   1:  PR[GP1:91,2] = PR[GP1:90,2] + -1.651;
   1:L PR[91] R[100]mm/sec CNT100;
   1:  PR[GP1:91,1] = PR[GP1:90,1] + -34.835;
   1:  PR[GP1:91,2] = PR[GP1:90,2] + -4.892;
   1:L PR[91] R[100]mm/sec CNT100;
   1:  PR[GP1:91,1] = PR[GP1:90,1] + -34.523;
   1:  PR[GP1:91,2] = PR[GP1:90,2] + -6.094;
   1:L PR[91] R[100]mm/sec CNT100;
   1:  PR[GP1:91,1] = PR[GP1:90,1] + -33.966;
   1:  PR[GP1:91,2] = PR[GP1:90,2] + -7.337;
   1:L PR[91] R[100]mm/sec CNT100;
   1:  PR[GP1:91,1] = PR[GP1:90,1] + -32.585;
   1:  PR[GP1:91,2] = PR[GP1:90,2] + -10.486;
   1:L PR[91] R[100]mm/sec CNT100;
   1:  PR[GP1:91,1] = PR[GP1:90,1] + -31.931;
   1:  PR[GP1:91,2] = PR[GP1:90,2] + -11.478;
   1:L PR[91] R[100]mm/sec CNT100;
   1:  PR[GP1:91,1] = PR[GP1:90,1] + -29.572;
   1:  PR[GP1:91,2] = PR[GP1:90,2] + -14.403;
   1:L PR[91] R[100]mm/sec CNT100;
   1:  PR[GP1:91,1] = PR[GP1:90,1] + -28.833;
   1:  PR[GP1:91,2] = PR[GP1:90,2] + -15.201;
   1:L PR[91] R[100]mm/sec CNT100;
   1:  PR[GP1:91,1] = PR[GP1:90,1] + -28.025;
   1:  PR[GP1:91,2] = PR[GP1:90,2] + -15.834;
   1:L PR[91] R[100]mm/sec CNT100;
   1:  PR[GP1:91,1] = PR[GP1:90,1] + -24.662;
   1:  PR[GP1:91,2] = PR[GP1:90,2] + -18.272;
   1:L PR[91] R[100]mm/sec CNT100;
   1:  PR[GP1:91,1] = PR[GP1:90,1] + -23.931;
   1:  PR[GP1:91,2] = PR[GP1:90,2] + -18.681;
   1:L PR[91] R[100]mm/sec CNT100;
   1:  PR[GP1:91,1] = PR[GP1:90,1] + -23.152;
   1:  PR[GP1:91,2] = PR[GP1:90,2] + -18.969;
   1:L PR[91] R[100]mm/sec CNT100;
   1:  PR[GP1:91,1] = PR[GP1:90,1] + -18.880;
   1:  PR[GP1:91,2] = PR[GP1:90,2] + -20.635;
   1:L PR[91] R[100]mm/sec CNT100;
   1:  PR[GP1:91,1] = PR[GP1:90,1] + -18.320;
   1:  PR[GP1:91,2] = PR[GP1:90,2] + -20.751;
   1:L PR[91] R[100]mm/sec CNT100;
   1:  PR[GP1:91,1] = PR[GP1:90,1] + -13.243;
   1:  PR[GP1:91,2] = PR[GP1:90,2] + -21.342;
   1:L PR[91] R[100]mm/sec CNT100;
   1:  PR[GP1:91,1] = PR[GP1:90,1] + -12.848;
   1:  PR[GP1:91,2] = PR[GP1:90,2] + -21.363;
   1:L PR[91] R[100]mm/sec CNT100;
   1:  PR[GP1:91,1] = PR[GP1:90,1] + -12.498;
   1:  PR[GP1:91,2] = PR[GP1:90,2] + -21.328;
   1:L PR[91] R[100]mm/sec CNT100;
   1:  PR[GP1:91,1] = PR[GP1:90,1] + -7.066;
   1:  PR[GP1:91,2] = PR[GP1:90,2] + -20.567;
   1:L PR[91] R[100]mm/sec CNT100;
   1:  PR[GP1:91,1] = PR[GP1:90,1] + -6.974;
   1:  PR[GP1:91,2] = PR[GP1:90,2] + -20.544;
   1:L PR[91] R[100]mm/sec CNT100;
   1:  PR[GP1:91,1] = PR[GP1:90,1] + -1.723;
   1:  PR[GP1:91,2] = PR[GP1:90,2] + -18.303;
   1:L PR[91] R[100]mm/sec CNT100;
   1:  PR[GP1:91,1] = PR[GP1:90,1] + -1.227;
   1:  PR[GP1:91,2] = PR[GP1:90,2] + -18.103;
   1:L PR[91] R[100]mm/sec CNT100;
   1:  PR[GP1:91,1] = PR[GP1:90,1] + -0.702;
   1:  PR[GP1:91,2] = PR[GP1:90,2] + -17.952;
   1:L PR[91] R[100]mm/sec CNT100;
   1:  PR[GP1:91,1] = PR[GP1:90,1] + 0.096;
   1:  PR[GP1:91,2] = PR[GP1:90,2] + -17.623;
   1:L PR[91] R[100]mm/sec CNT100;
   1:  PR[GP1:91,1] = PR[GP1:90,1] + 1.055;
   1:  PR[GP1:91,2] = PR[GP1:90,2] + -17.917;
   1:L PR[91] R[100]mm/sec CNT100;
   1:  PR[GP1:91,1] = PR[GP1:90,1] + 1.526;
   1:  PR[GP1:91,2] = PR[GP1:90,2] + -18.164;
   1:L PR[91] R[100]mm/sec CNT100;
   1:  PR[GP1:91,1] = PR[GP1:90,1] + 7.126;
   1:  PR[GP1:91,2] = PR[GP1:90,2] + -20.540;
   1:L PR[91] R[100]mm/sec CNT100;
   1:  PR[GP1:91,1] = PR[GP1:90,1] + 7.196;
   1:  PR[GP1:91,2] = PR[GP1:90,2] + -20.559;
   1:L PR[91] R[100]mm/sec CNT100;
   1:  PR[GP1:91,1] = PR[GP1:90,1] + 7.432;
   1:  PR[GP1:91,2] = PR[GP1:90,2] + -20.583;
   1:L PR[91] R[100]mm/sec CNT100;
   1:  PR[GP1:91,1] = PR[GP1:90,1] + 13.029;
   1:  PR[GP1:91,2] = PR[GP1:90,2] + -21.362;
   1:L PR[91] R[100]mm/sec CNT100;
   1:  PR[GP1:91,1] = PR[GP1:90,1] + 13.393;
   1:  PR[GP1:91,2] = PR[GP1:90,2] + -21.343;
   1:L PR[91] R[100]mm/sec CNT100;
   1:  PR[GP1:91,1] = PR[GP1:90,1] + 18.470;
   1:  PR[GP1:91,2] = PR[GP1:90,2] + -20.751;
   1:L PR[91] R[100]mm/sec CNT100;
   1:  PR[GP1:91,1] = PR[GP1:90,1] + 19.041;
   1:  PR[GP1:91,2] = PR[GP1:90,2] + -20.633;
   1:L PR[91] R[100]mm/sec CNT100;
   1:  PR[GP1:91,1] = PR[GP1:90,1] + 19.722;
   1:  PR[GP1:91,2] = PR[GP1:90,2] + -20.382;
   1:L PR[91] R[100]mm/sec CNT100;
   1:  PR[GP1:91,1] = PR[GP1:90,1] + 24.072;
   1:  PR[GP1:91,2] = PR[GP1:90,2] + -18.690;
   1:L PR[91] R[100]mm/sec CNT100;
   1:  PR[GP1:91,1] = PR[GP1:90,1] + 24.789;
   1:  PR[GP1:91,2] = PR[GP1:90,2] + -18.291;
   1:L PR[91] R[100]mm/sec CNT100;
   1:  PR[GP1:91,1] = PR[GP1:90,1] + 25.600;
   1:  PR[GP1:91,2] = PR[GP1:90,2] + -17.662;
   1:L PR[91] R[100]mm/sec CNT100;
   1:  PR[GP1:91,1] = PR[GP1:90,1] + 28.990;
   1:  PR[GP1:91,2] = PR[GP1:90,2] + -15.200;
   1:L PR[91] R[100]mm/sec CNT100;
   1:  PR[GP1:91,1] = PR[GP1:90,1] + 29.712;
   1:  PR[GP1:91,2] = PR[GP1:90,2] + -14.420;
   1:L PR[91] R[100]mm/sec CNT100;
   1:  PR[GP1:91,1] = PR[GP1:90,1] + 32.073;
   1:  PR[GP1:91,2] = PR[GP1:90,2] + -11.489;
   1:L PR[91] R[100]mm/sec CNT100;
   1:  PR[GP1:91,1] = PR[GP1:90,1] + 32.740;
   1:  PR[GP1:91,2] = PR[GP1:90,2] + -10.480;
   1:L PR[91] R[100]mm/sec CNT100;
   1:  PR[GP1:91,1] = PR[GP1:90,1] + 33.295;
   1:  PR[GP1:91,2] = PR[GP1:90,2] + -9.259;
   1:L PR[91] R[100]mm/sec CNT100;
   1:  PR[GP1:91,1] = PR[GP1:90,1] + 34.672;
   1:  PR[GP1:91,2] = PR[GP1:90,2] + -6.135;
   1:L PR[91] R[100]mm/sec CNT100;
   1:  PR[GP1:91,1] = PR[GP1:90,1] + 34.975;
   1:  PR[GP1:91,2] = PR[GP1:90,2] + -4.983;
   1:L PR[91] R[100]mm/sec CNT100;
   1:  PR[GP1:91,1] = PR[GP1:90,1] + 35.092;
   1:  PR[GP1:91,2] = PR[GP1:90,2] + -3.555;
   1:L PR[91] R[100]mm/sec CNT100;
   1:  PR[GP1:91,1] = PR[GP1:90,1] + 35.547;
   1:  PR[GP1:91,2] = PR[GP1:90,2] + -0.271;
   1:L PR[91] R[100]mm/sec CNT100;
   1:  PR[GP1:91,1] = PR[GP1:90,1] + 35.437;
   1:  PR[GP1:91,2] = PR[GP1:90,2] + 1.070;
   1:L PR[91] R[100]mm/sec CNT100;
   1:  PR[GP1:91,1] = PR[GP1:90,1] + 34.986;
   1:  PR[GP1:91,2] = PR[GP1:90,2] + 4.315;
   1:L PR[91] R[100]mm/sec CNT100;
   1:  PR[GP1:91,1] = PR[GP1:90,1] + 34.676;
   1:  PR[GP1:91,2] = PR[GP1:90,2] + 5.499;
   1:L PR[91] R[100]mm/sec CNT100;
   1:  PR[GP1:91,1] = PR[GP1:90,1] + 34.119;
   1:  PR[GP1:91,2] = PR[GP1:90,2] + 6.723;
   1:L PR[91] R[100]mm/sec CNT100;
   1:  PR[GP1:91,1] = PR[GP1:90,1] + 32.741;
   1:  PR[GP1:91,2] = PR[GP1:90,2] + 9.856;
   1:L PR[91] R[100]mm/sec CNT100;
   1:  PR[GP1:91,1] = PR[GP1:90,1] + 32.078;
   1:  PR[GP1:91,2] = PR[GP1:90,2] + 10.857;
   1:L PR[91] R[100]mm/sec CNT100;
   1:  PR[GP1:91,1] = PR[GP1:90,1] + 29.723;
   1:  PR[GP1:91,2] = PR[GP1:90,2] + 13.786;
   1:L PR[91] R[100]mm/sec CNT100;
   1:  PR[GP1:91,1] = PR[GP1:90,1] + 28.984;
   1:  PR[GP1:91,2] = PR[GP1:90,2] + 14.583;
   1:L PR[91] R[100]mm/sec CNT100;
   1:  PR[GP1:91,1] = PR[GP1:90,1] + 28.182;
   1:  PR[GP1:91,2] = PR[GP1:90,2] + 15.208;
   1:L PR[91] R[100]mm/sec CNT100;
   1:  PR[GP1:91,1] = PR[GP1:90,1] + 24.828;
   1:  PR[GP1:91,2] = PR[GP1:90,2] + 17.645;
   1:L PR[91] R[100]mm/sec CNT100;
   1:  PR[GP1:91,1] = PR[GP1:90,1] + 24.103;
   1:  PR[GP1:91,2] = PR[GP1:90,2] + 18.049;
   1:L PR[91] R[100]mm/sec CNT100;
   1:  PR[GP1:91,1] = PR[GP1:90,1] + 23.320;
   1:  PR[GP1:91,2] = PR[GP1:90,2] + 18.337;
   1:L PR[91] R[100]mm/sec CNT100;
   1:  PR[GP1:91,1] = PR[GP1:90,1] + 19.058;
   1:  PR[GP1:91,2] = PR[GP1:90,2] + 20.004;
   1:L PR[91] R[100]mm/sec CNT100;
   1:  PR[GP1:91,1] = PR[GP1:90,1] + 18.498;
   1:  PR[GP1:91,2] = PR[GP1:90,2] + 20.120;
   1:L PR[91] R[100]mm/sec CNT100;
   1:  PR[GP1:91,1] = PR[GP1:90,1] + 13.433;
   1:  PR[GP1:91,2] = PR[GP1:90,2] + 20.719;
   1:L PR[91] R[100]mm/sec CNT100;
   1:  PR[GP1:91,1] = PR[GP1:90,1] + 13.042;
   1:  PR[GP1:91,2] = PR[GP1:90,2] + 20.740;
   1:L PR[91] R[100]mm/sec CNT100;
   1:  PR[GP1:91,1] = PR[GP1:90,1] + 12.690;
   1:  PR[GP1:91,2] = PR[GP1:90,2] + 20.704;
   1:L PR[91] R[100]mm/sec CNT100;
   1:  PR[GP1:91,1] = PR[GP1:90,1] + 7.269;
   1:  PR[GP1:91,2] = PR[GP1:90,2] + 19.954;
   1:L PR[91] R[100]mm/sec CNT100;
   1:  PR[GP1:91,1] = PR[GP1:90,1] + 7.171;
   1:  PR[GP1:91,2] = PR[GP1:90,2] + 19.929;
   1:L PR[91] R[100]mm/sec CNT100;
   1:  PR[GP1:91,1] = PR[GP1:90,1] + 1.706;
   1:  PR[GP1:91,2] = PR[GP1:90,2] + 17.641;
   1:L PR[91] R[100]mm/sec CNT100;
   1:  PR[GP1:91,1] = PR[GP1:90,1] + 1.616;
   1:  PR[GP1:91,2] = PR[GP1:90,2] + 17.580;
   1:L PR[91] R[100]mm/sec CNT100;
   1:  PR[GP1:91,1] = PR[GP1:90,1] + 1.237;
   1:  PR[GP1:91,2] = PR[GP1:90,2] + 17.407;
   1:L PR[91] R[100]mm/sec CNT100;
   1:  PR[GP1:91,1] = PR[GP1:90,1] + 0.248;
   1:  PR[GP1:91,2] = PR[GP1:90,2] + 17.007;
   1:L PR[91] R[100]mm/sec CNT100;
   1:  PR[91] = PR[90];
   1:  PR[GP1:91,1] = PR[GP1:90,1] + -1.228;
   1:  PR[GP1:91,2] = PR[GP1:90,2] + 17.668;
   1:  PR[GP1:91,3] = PR[GP1:90,3] + 40.565;
   1:L PR[91] R[100]mm/sec CNT100;
   1:  PR[GP1:91,1] = PR[GP1:90,1] + -1.389;
   1:  PR[GP1:91,2] = PR[GP1:90,2] + 17.767;
   1:L PR[91] R[100]mm/sec CNT100;
   1:  PR[GP1:91,1] = PR[GP1:90,1] + -3.118;
   1:  PR[GP1:91,2] = PR[GP1:90,2] + 18.458;
   1:L PR[91] R[100]mm/sec CNT100;
   1:  PR[GP1:91,1] = PR[GP1:90,1] + -6.808;
   1:  PR[GP1:91,2] = PR[GP1:90,2] + 20.004;
   1:L PR[91] R[100]mm/sec CNT100;
   1:  PR[GP1:91,1] = PR[GP1:90,1] + -12.690;
   1:  PR[GP1:91,2] = PR[GP1:90,2] + 20.802;
   1:L PR[91] R[100]mm/sec CNT100;
   1:  PR[GP1:91,1] = PR[GP1:90,1] + -12.917;
   1:  PR[GP1:91,2] = PR[GP1:90,2] + 20.790;
   1:L PR[91] R[100]mm/sec CNT100;
   1:  PR[GP1:91,1] = PR[GP1:90,1] + -18.224;
   1:  PR[GP1:91,2] = PR[GP1:90,2] + 20.163;
   1:L PR[91] R[100]mm/sec CNT100;
   1:  PR[GP1:91,1] = PR[GP1:90,1] + -18.664;
   1:  PR[GP1:91,2] = PR[GP1:90,2] + 20.071;
   1:L PR[91] R[100]mm/sec CNT100;
   1:  PR[GP1:91,1] = PR[GP1:90,1] + -19.201;
   1:  PR[GP1:91,2] = PR[GP1:90,2] + 19.872;
   1:L PR[91] R[100]mm/sec CNT100;
   1:  PR[GP1:91,1] = PR[GP1:90,1] + -23.778;
   1:  PR[GP1:91,2] = PR[GP1:90,2] + 18.083;
   1:L PR[91] R[100]mm/sec CNT100;
   1:  PR[GP1:91,1] = PR[GP1:90,1] + -24.373;
   1:  PR[GP1:91,2] = PR[GP1:90,2] + 17.749;
   1:L PR[91] R[100]mm/sec CNT100;
   1:  PR[GP1:91,1] = PR[GP1:90,1] + -25.068;
   1:  PR[GP1:91,2] = PR[GP1:90,2] + 17.208;
   1:L PR[91] R[100]mm/sec CNT100;
   1:  PR[GP1:91,1] = PR[GP1:90,1] + -28.665;
   1:  PR[GP1:91,2] = PR[GP1:90,2] + 14.588;
   1:L PR[91] R[100]mm/sec CNT100;
   1:  PR[GP1:91,1] = PR[GP1:90,1] + -29.286;
   1:  PR[GP1:91,2] = PR[GP1:90,2] + 13.917;
   1:L PR[91] R[100]mm/sec CNT100;
   1:  PR[GP1:91,1] = PR[GP1:90,1] + -31.800;
   1:  PR[GP1:91,2] = PR[GP1:90,2] + 10.796;
   1:L PR[91] R[100]mm/sec CNT100;
   1:  PR[GP1:91,1] = PR[GP1:90,1] + -32.375;
   1:  PR[GP1:91,2] = PR[GP1:90,2] + 9.922;
   1:L PR[91] R[100]mm/sec CNT100;
   1:  PR[GP1:91,1] = PR[GP1:90,1] + -34.349;
   1:  PR[GP1:91,2] = PR[GP1:90,2] + 5.445;
   1:L PR[91] R[100]mm/sec CNT100;
   1:  PR[GP1:91,1] = PR[GP1:90,1] + -34.615;
   1:  PR[GP1:91,2] = PR[GP1:90,2] + 4.416;
   1:L PR[91] R[100]mm/sec CNT100;
   1:  PR[GP1:91,1] = PR[GP1:90,1] + -34.715;
   1:  PR[GP1:91,2] = PR[GP1:90,2] + 3.173;
   1:L PR[91] R[100]mm/sec CNT100;
   1:  PR[GP1:91,1] = PR[GP1:90,1] + -35.204;
   1:  PR[GP1:91,2] = PR[GP1:90,2] + -0.354;
   1:L PR[91] R[100]mm/sec CNT100;
   1:  PR[GP1:91,1] = PR[GP1:90,1] + -35.112;
   1:  PR[GP1:91,2] = PR[GP1:90,2] + -1.511;
   1:L PR[91] R[100]mm/sec CNT100;
   1:  PR[GP1:91,1] = PR[GP1:90,1] + -34.625;
   1:  PR[GP1:91,2] = PR[GP1:90,2] + -5.003;
   1:L PR[91] R[100]mm/sec CNT100;
   1:  PR[GP1:91,1] = PR[GP1:90,1] + -34.349;
   1:  PR[GP1:91,2] = PR[GP1:90,2] + -6.069;
   1:L PR[91] R[100]mm/sec CNT100;
   1:  PR[GP1:91,1] = PR[GP1:90,1] + -33.850;
   1:  PR[GP1:91,2] = PR[GP1:90,2] + -7.180;
   1:L PR[91] R[100]mm/sec CNT100;
   1:  PR[GP1:91,1] = PR[GP1:90,1] + -32.369;
   1:  PR[GP1:91,2] = PR[GP1:90,2] + -10.555;
   1:L PR[91] R[100]mm/sec CNT100;
   1:  PR[GP1:91,1] = PR[GP1:90,1] + -31.795;
   1:  PR[GP1:91,2] = PR[GP1:90,2] + -11.428;
   1:L PR[91] R[100]mm/sec CNT100;
   1:  PR[GP1:91,1] = PR[GP1:90,1] + -29.275;
   1:  PR[GP1:91,2] = PR[GP1:90,2] + -14.552;
   1:L PR[91] R[100]mm/sec CNT100;
   1:  PR[GP1:91,1] = PR[GP1:90,1] + -28.636;
   1:  PR[GP1:91,2] = PR[GP1:90,2] + -15.242;
   1:L PR[91] R[100]mm/sec CNT100;
   1:  PR[GP1:91,1] = PR[GP1:90,1] + -27.936;
   1:  PR[GP1:91,2] = PR[GP1:90,2] + -15.790;
   1:L PR[91] R[100]mm/sec CNT100;
   1:  PR[GP1:91,1] = PR[GP1:90,1] + -24.373;
   1:  PR[GP1:91,2] = PR[GP1:90,2] + -18.373;
   1:L PR[91] R[100]mm/sec CNT100;
   1:  PR[GP1:91,1] = PR[GP1:90,1] + -23.769;
   1:  PR[GP1:91,2] = PR[GP1:90,2] + -18.711;
   1:L PR[91] R[100]mm/sec CNT100;
   1:  PR[GP1:91,1] = PR[GP1:90,1] + -23.112;
   1:  PR[GP1:91,2] = PR[GP1:90,2] + -18.954;
   1:L PR[91] R[100]mm/sec CNT100;
   1:  PR[GP1:91,1] = PR[GP1:90,1] + -18.620;
   1:  PR[GP1:91,2] = PR[GP1:90,2] + -20.706;
   1:L PR[91] R[100]mm/sec CNT100;
   1:  PR[GP1:91,1] = PR[GP1:90,1] + -18.194;
   1:  PR[GP1:91,2] = PR[GP1:90,2] + -20.794;
   1:L PR[91] R[100]mm/sec CNT100;
   1:  PR[GP1:91,1] = PR[GP1:90,1] + -12.873;
   1:  PR[GP1:91,2] = PR[GP1:90,2] + -21.414;
   1:L PR[91] R[100]mm/sec CNT100;
   1:  PR[GP1:91,1] = PR[GP1:90,1] + -12.622;
   1:  PR[GP1:91,2] = PR[GP1:90,2] + -21.427;
   1:L PR[91] R[100]mm/sec CNT100;
   1:  PR[GP1:91,1] = PR[GP1:90,1] + -12.399;
   1:  PR[GP1:91,2] = PR[GP1:90,2] + -21.404;
   1:L PR[91] R[100]mm/sec CNT100;
   1:  PR[GP1:91,1] = PR[GP1:90,1] + -6.761;
   1:  PR[GP1:91,2] = PR[GP1:90,2] + -20.615;
   1:L PR[91] R[100]mm/sec CNT100;
   1:  PR[GP1:91,1] = PR[GP1:90,1] + -4.016;
   1:  PR[GP1:91,2] = PR[GP1:90,2] + -19.444;
   1:L PR[91] R[100]mm/sec CNT100;
   1:  PR[GP1:91,1] = PR[GP1:90,1] + -1.135;
   1:  PR[GP1:91,2] = PR[GP1:90,2] + -18.283;
   1:L PR[91] R[100]mm/sec CNT100;
   1:  PR[GP1:91,1] = PR[GP1:90,1] + -0.880;
   1:  PR[GP1:91,2] = PR[GP1:90,2] + -18.239;
   1:L PR[91] R[100]mm/sec CNT100;
   1:  PR[GP1:91,1] = PR[GP1:90,1] + -0.618;
   1:  PR[GP1:91,2] = PR[GP1:90,2] + -18.162;
   1:L PR[91] R[100]mm/sec CNT100;
   1:  PR[GP1:91,1] = PR[GP1:90,1] + 0.116;
   1:  PR[GP1:91,2] = PR[GP1:90,2] + -17.860;
   1:L PR[91] R[100]mm/sec CNT100;
   1:  PR[GP1:91,1] = PR[GP1:90,1] + 1.110;
   1:  PR[GP1:91,2] = PR[GP1:90,2] + -18.164;
   1:L PR[91] R[100]mm/sec CNT100;
   1:  PR[GP1:91,1] = PR[GP1:90,1] + 1.497;
   1:  PR[GP1:91,2] = PR[GP1:90,2] + -18.367;
   1:L PR[91] R[100]mm/sec CNT100;
   1:  PR[GP1:91,1] = PR[GP1:90,1] + 4.169;
   1:  PR[GP1:91,2] = PR[GP1:90,2] + -19.443;
   1:L PR[91] R[100]mm/sec CNT100;
   1:  PR[GP1:91,1] = PR[GP1:90,1] + 6.913;
   1:  PR[GP1:91,2] = PR[GP1:90,2] + -20.612;
   1:L PR[91] R[100]mm/sec CNT100;
   1:  PR[GP1:91,1] = PR[GP1:90,1] + 12.803;
   1:  PR[GP1:91,2] = PR[GP1:90,2] + -21.426;
   1:L PR[91] R[100]mm/sec CNT100;
   1:  PR[GP1:91,1] = PR[GP1:90,1] + 13.025;
   1:  PR[GP1:91,2] = PR[GP1:90,2] + -21.414;
   1:L PR[91] R[100]mm/sec CNT100;
   1:  PR[GP1:91,1] = PR[GP1:90,1] + 18.344;
   1:  PR[GP1:91,2] = PR[GP1:90,2] + -20.795;
   1:L PR[91] R[100]mm/sec CNT100;
   1:  PR[GP1:91,1] = PR[GP1:90,1] + 18.782;
   1:  PR[GP1:91,2] = PR[GP1:90,2] + -20.704;
   1:L PR[91] R[100]mm/sec CNT100;
   1:  PR[GP1:91,1] = PR[GP1:90,1] + 19.320;
   1:  PR[GP1:91,2] = PR[GP1:90,2] + -20.505;
   1:L PR[91] R[100]mm/sec CNT100;
   1:  PR[GP1:91,1] = PR[GP1:90,1] + 23.910;
   1:  PR[GP1:91,2] = PR[GP1:90,2] + -18.721;
   1:L PR[91] R[100]mm/sec CNT100;
   1:  PR[GP1:91,1] = PR[GP1:90,1] + 24.501;
   1:  PR[GP1:91,2] = PR[GP1:90,2] + -18.391;
   1:L PR[91] R[100]mm/sec CNT100;
   1:  PR[GP1:91,1] = PR[GP1:90,1] + 25.190;
   1:  PR[GP1:91,2] = PR[GP1:90,2] + -17.858;
   1:L PR[91] R[100]mm/sec CNT100;
   1:  PR[GP1:91,1] = PR[GP1:90,1] + 28.795;
   1:  PR[GP1:91,2] = PR[GP1:90,2] + -15.239;
   1:L PR[91] R[100]mm/sec CNT100;
   1:  PR[GP1:91,1] = PR[GP1:90,1] + 29.417;
   1:  PR[GP1:91,2] = PR[GP1:90,2] + -14.567;
   1:L PR[91] R[100]mm/sec CNT100;
   1:  PR[GP1:91,1] = PR[GP1:90,1] + 31.939;
   1:  PR[GP1:91,2] = PR[GP1:90,2] + -11.436;
   1:L PR[91] R[100]mm/sec CNT100;
   1:  PR[GP1:91,1] = PR[GP1:90,1] + 32.526;
   1:  PR[GP1:91,2] = PR[GP1:90,2] + -10.549;
   1:L PR[91] R[100]mm/sec CNT100;
   1:  PR[GP1:91,1] = PR[GP1:90,1] + 33.017;
   1:  PR[GP1:91,2] = PR[GP1:90,2] + -9.467;
   1:L PR[91] R[100]mm/sec CNT100;
   1:  PR[GP1:91,1] = PR[GP1:90,1] + 34.498;
   1:  PR[GP1:91,2] = PR[GP1:90,2] + -6.107;
   1:L PR[91] R[100]mm/sec CNT100;
   1:  PR[GP1:91,1] = PR[GP1:90,1] + 34.765;
   1:  PR[GP1:91,2] = PR[GP1:90,2] + -5.091;
   1:L PR[91] R[100]mm/sec CNT100;
   1:  PR[GP1:91,1] = PR[GP1:90,1] + 34.870;
   1:  PR[GP1:91,2] = PR[GP1:90,2] + -3.810;
   1:L PR[91] R[100]mm/sec CNT100;
   1:  PR[GP1:91,1] = PR[GP1:90,1] + 35.360;
   1:  PR[GP1:91,2] = PR[GP1:90,2] + -0.271;
   1:L PR[91] R[100]mm/sec CNT100;
   1:  PR[GP1:91,1] = PR[GP1:90,1] + 35.263;
   1:  PR[GP1:91,2] = PR[GP1:90,2] + 0.927;
   1:L PR[91] R[100]mm/sec CNT100;
   1:  PR[GP1:91,1] = PR[GP1:90,1] + 34.777;
   1:  PR[GP1:91,2] = PR[GP1:90,2] + 4.423;
   1:L PR[91] R[100]mm/sec CNT100;
   1:  PR[GP1:91,1] = PR[GP1:90,1] + 34.502;
   1:  PR[GP1:91,2] = PR[GP1:90,2] + 5.471;
   1:L PR[91] R[100]mm/sec CNT100;
   1:  PR[GP1:91,1] = PR[GP1:90,1] + 34.004;
   1:  PR[GP1:91,2] = PR[GP1:90,2] + 6.565;
   1:L PR[91] R[100]mm/sec CNT100;
   1:  PR[GP1:91,1] = PR[GP1:90,1] + 32.526;
   1:  PR[GP1:91,2] = PR[GP1:90,2] + 9.924;
   1:L PR[91] R[100]mm/sec CNT100;
   1:  PR[GP1:91,1] = PR[GP1:90,1] + 31.943;
   1:  PR[GP1:91,2] = PR[GP1:90,2] + 10.804;
   1:L PR[91] R[100]mm/sec CNT100;
   1:  PR[GP1:91,1] = PR[GP1:90,1] + 29.429;
   1:  PR[GP1:91,2] = PR[GP1:90,2] + 13.932;
   1:L PR[91] R[100]mm/sec CNT100;
   1:  PR[GP1:91,1] = PR[GP1:90,1] + 28.790;
   1:  PR[GP1:91,2] = PR[GP1:90,2] + 14.621;
   1:L PR[91] R[100]mm/sec CNT100;
   1:  PR[GP1:91,1] = PR[GP1:90,1] + 28.095;
   1:  PR[GP1:91,2] = PR[GP1:90,2] + 15.163;
   1:L PR[91] R[100]mm/sec CNT100;
   1:  PR[GP1:91,1] = PR[GP1:90,1] + 24.541;
   1:  PR[GP1:91,2] = PR[GP1:90,2] + 17.745;
   1:L PR[91] R[100]mm/sec CNT100;
   1:  PR[GP1:91,1] = PR[GP1:90,1] + 23.942;
   1:  PR[GP1:91,2] = PR[GP1:90,2] + 18.079;
   1:L PR[91] R[100]mm/sec CNT100;
   1:  PR[GP1:91,1] = PR[GP1:90,1] + 23.282;
   1:  PR[GP1:91,2] = PR[GP1:90,2] + 18.322;
   1:L PR[91] R[100]mm/sec CNT100;
   1:  PR[GP1:91,1] = PR[GP1:90,1] + 18.801;
   1:  PR[GP1:91,2] = PR[GP1:90,2] + 20.075;
   1:L PR[91] R[100]mm/sec CNT100;
   1:  PR[GP1:91,1] = PR[GP1:90,1] + 18.374;
   1:  PR[GP1:91,2] = PR[GP1:90,2] + 20.163;
   1:L PR[91] R[100]mm/sec CNT100;
   1:  PR[GP1:91,1] = PR[GP1:90,1] + 13.067;
   1:  PR[GP1:91,2] = PR[GP1:90,2] + 20.791;
   1:L PR[91] R[100]mm/sec CNT100;
   1:  PR[GP1:91,1] = PR[GP1:90,1] + 12.818;
   1:  PR[GP1:91,2] = PR[GP1:90,2] + 20.804;
   1:L PR[91] R[100]mm/sec CNT100;
   1:  PR[GP1:91,1] = PR[GP1:90,1] + 12.593;
   1:  PR[GP1:91,2] = PR[GP1:90,2] + 20.781;
   1:L PR[91] R[100]mm/sec CNT100;
   1:  PR[GP1:91,1] = PR[GP1:90,1] + 6.961;
   1:  PR[GP1:91,2] = PR[GP1:90,2] + 20.002;
   1:L PR[91] R[100]mm/sec CNT100;
   1:  PR[GP1:91,1] = PR[GP1:90,1] + 3.272;
   1:  PR[GP1:91,2] = PR[GP1:90,2] + 18.458;
   1:L PR[91] R[100]mm/sec CNT100;
   1:  PR[GP1:91,1] = PR[GP1:90,1] + 1.382;
   1:  PR[GP1:91,2] = PR[GP1:90,2] + 17.706;
   1:L PR[91] R[100]mm/sec CNT100;
   1:  PR[GP1:91,1] = PR[GP1:90,1] + 0.282;
   1:  PR[GP1:91,2] = PR[GP1:90,2] + 17.240;
   1:L PR[91] R[100]mm/sec CNT100;
   1:  PR[91] = PR[90];
   1:  PR[GP1:91,1] = PR[GP1:90,1] + -1.166;
   1:  PR[GP1:91,2] = PR[GP1:90,2] + 17.893;
   1:  PR[GP1:91,3] = PR[GP1:90,3] + 41.175;
   1:L PR[91] R[100]mm/sec CNT100;
   1:  PR[GP1:91,1] = PR[GP1:90,1] + -6.558;
   1:  PR[GP1:91,2] = PR[GP1:90,2] + 20.060;
   1:L PR[91] R[100]mm/sec CNT100;
   1:  PR[GP1:91,1] = PR[GP1:90,1] + -12.467;
   1:  PR[GP1:91,2] = PR[GP1:90,2] + 20.866;
   1:L PR[91] R[100]mm/sec CNT100;
   1:  PR[GP1:91,1] = PR[GP1:90,1] + -12.549;
   1:  PR[GP1:91,2] = PR[GP1:90,2] + 20.862;
   1:L PR[91] R[100]mm/sec CNT100;
   1:  PR[GP1:91,1] = PR[GP1:90,1] + -18.099;
   1:  PR[GP1:91,2] = PR[GP1:90,2] + 20.205;
   1:L PR[91] R[100]mm/sec CNT100;
   1:  PR[GP1:91,1] = PR[GP1:90,1] + -18.406;
   1:  PR[GP1:91,2] = PR[GP1:90,2] + 20.142;
   1:L PR[91] R[100]mm/sec CNT100;
   1:  PR[GP1:91,1] = PR[GP1:90,1] + -18.800;
   1:  PR[GP1:91,2] = PR[GP1:90,2] + 19.995;
   1:L PR[91] R[100]mm/sec CNT100;
   1:  PR[GP1:91,1] = PR[GP1:90,1] + -23.616;
   1:  PR[GP1:91,2] = PR[GP1:90,2] + 18.113;
   1:L PR[91] R[100]mm/sec CNT100;
   1:  PR[GP1:91,1] = PR[GP1:90,1] + -24.085;
   1:  PR[GP1:91,2] = PR[GP1:90,2] + 17.850;
   1:L PR[91] R[100]mm/sec CNT100;
   1:  PR[GP1:91,1] = PR[GP1:90,1] + -24.657;
   1:  PR[GP1:91,2] = PR[GP1:90,2] + 17.405;
   1:L PR[91] R[100]mm/sec CNT100;
   1:  PR[GP1:91,1] = PR[GP1:90,1] + -28.469;
   1:  PR[GP1:91,2] = PR[GP1:90,2] + 14.628;
   1:L PR[91] R[100]mm/sec CNT100;
   1:  PR[GP1:91,1] = PR[GP1:90,1] + -28.991;
   1:  PR[GP1:91,2] = PR[GP1:90,2] + 14.065;
   1:L PR[91] R[100]mm/sec CNT100;
   1:  PR[GP1:91,1] = PR[GP1:90,1] + -31.665;
   1:  PR[GP1:91,2] = PR[GP1:90,2] + 10.745;
   1:L PR[91] R[100]mm/sec CNT100;
   1:  PR[GP1:91,1] = PR[GP1:90,1] + -32.160;
   1:  PR[GP1:91,2] = PR[GP1:90,2] + 9.991;
   1:L PR[91] R[100]mm/sec CNT100;
   1:  PR[GP1:91,1] = PR[GP1:90,1] + -34.174;
   1:  PR[GP1:91,2] = PR[GP1:90,2] + 5.420;
   1:L PR[91] R[100]mm/sec CNT100;
   1:  PR[GP1:91,1] = PR[GP1:90,1] + -34.405;
   1:  PR[GP1:91,2] = PR[GP1:90,2] + 4.527;
   1:L PR[91] R[100]mm/sec CNT100;
   1:  PR[GP1:91,1] = PR[GP1:90,1] + -34.493;
   1:  PR[GP1:91,2] = PR[GP1:90,2] + 3.428;
   1:L PR[91] R[100]mm/sec CNT100;
   1:  PR[GP1:91,1] = PR[GP1:90,1] + -35.017;
   1:  PR[GP1:91,2] = PR[GP1:90,2] + -0.354;
   1:L PR[91] R[100]mm/sec CNT100;
   1:  PR[GP1:91,1] = PR[GP1:90,1] + -34.936;
   1:  PR[GP1:91,2] = PR[GP1:90,2] + -1.372;
   1:L PR[91] R[100]mm/sec CNT100;
   1:  PR[GP1:91,1] = PR[GP1:90,1] + -34.414;
   1:  PR[GP1:91,2] = PR[GP1:90,2] + -5.115;
   1:L PR[91] R[100]mm/sec CNT100;
   1:  PR[GP1:91,1] = PR[GP1:90,1] + -34.174;
   1:  PR[GP1:91,2] = PR[GP1:90,2] + -6.044;
   1:L PR[91] R[100]mm/sec CNT100;
   1:  PR[GP1:91,1] = PR[GP1:90,1] + -33.734;
   1:  PR[GP1:91,2] = PR[GP1:90,2] + -7.023;
   1:L PR[91] R[100]mm/sec CNT100;
   1:  PR[GP1:91,1] = PR[GP1:90,1] + -32.154;
   1:  PR[GP1:91,2] = PR[GP1:90,2] + -10.625;
   1:L PR[91] R[100]mm/sec CNT100;
   1:  PR[GP1:91,1] = PR[GP1:90,1] + -31.659;
   1:  PR[GP1:91,2] = PR[GP1:90,2] + -11.377;
   1:L PR[91] R[100]mm/sec CNT100;
   1:  PR[GP1:91,1] = PR[GP1:90,1] + -28.978;
   1:  PR[GP1:91,2] = PR[GP1:90,2] + -14.700;
   1:L PR[91] R[100]mm/sec CNT100;
   1:  PR[GP1:91,1] = PR[GP1:90,1] + -28.439;
   1:  PR[GP1:91,2] = PR[GP1:90,2] + -15.283;
   1:L PR[91] R[100]mm/sec CNT100;
   1:  PR[GP1:91,1] = PR[GP1:90,1] + -27.847;
   1:  PR[GP1:91,2] = PR[GP1:90,2] + -15.746;
   1:L PR[91] R[100]mm/sec CNT100;
   1:  PR[GP1:91,1] = PR[GP1:90,1] + -24.084;
   1:  PR[GP1:91,2] = PR[GP1:90,2] + -18.474;
   1:L PR[91] R[100]mm/sec CNT100;
   1:  PR[GP1:91,1] = PR[GP1:90,1] + -23.606;
   1:  PR[GP1:91,2] = PR[GP1:90,2] + -18.742;
   1:L PR[91] R[100]mm/sec CNT100;
   1:  PR[GP1:91,1] = PR[GP1:90,1] + -23.071;
   1:  PR[GP1:91,2] = PR[GP1:90,2] + -18.939;
   1:L PR[91] R[100]mm/sec CNT100;
   1:  PR[GP1:91,1] = PR[GP1:90,1] + -18.360;
   1:  PR[GP1:91,2] = PR[GP1:90,2] + -20.777;
   1:L PR[91] R[100]mm/sec CNT100;
   1:  PR[GP1:91,1] = PR[GP1:90,1] + -18.067;
   1:  PR[GP1:91,2] = PR[GP1:90,2] + -20.837;
   1:L PR[91] R[100]mm/sec CNT100;
   1:  PR[GP1:91,1] = PR[GP1:90,1] + -12.504;
   1:  PR[GP1:91,2] = PR[GP1:90,2] + -21.485;
   1:L PR[91] R[100]mm/sec CNT100;
   1:  PR[GP1:91,1] = PR[GP1:90,1] + -12.397;
   1:  PR[GP1:91,2] = PR[GP1:90,2] + -21.491;
   1:L PR[91] R[100]mm/sec CNT100;
   1:  PR[GP1:91,1] = PR[GP1:90,1] + -12.300;
   1:  PR[GP1:91,2] = PR[GP1:90,2] + -21.481;
   1:L PR[91] R[100]mm/sec CNT100;
   1:  PR[GP1:91,1] = PR[GP1:90,1] + -6.489;
   1:  PR[GP1:91,2] = PR[GP1:90,2] + -20.666;
   1:L PR[91] R[100]mm/sec CNT100;
   1:  PR[GP1:91,1] = PR[GP1:90,1] + -1.119;
   1:  PR[GP1:91,2] = PR[GP1:90,2] + -18.493;
   1:L PR[91] R[100]mm/sec CNT100;
   1:  PR[GP1:91,1] = PR[GP1:90,1] + -0.705;
   1:  PR[GP1:91,2] = PR[GP1:90,2] + -18.422;
   1:L PR[91] R[100]mm/sec CNT100;
   1:  PR[GP1:91,1] = PR[GP1:90,1] + -0.529;
   1:  PR[GP1:91,2] = PR[GP1:90,2] + -18.370;
   1:L PR[91] R[100]mm/sec CNT100;
   1:  PR[GP1:91,1] = PR[GP1:90,1] + 0.136;
   1:  PR[GP1:91,2] = PR[GP1:90,2] + -18.096;
   1:L PR[91] R[100]mm/sec CNT100;
   1:  PR[GP1:91,1] = PR[GP1:90,1] + 1.164;
   1:  PR[GP1:91,2] = PR[GP1:90,2] + -18.411;
   1:L PR[91] R[100]mm/sec CNT100;
   1:  PR[GP1:91,1] = PR[GP1:90,1] + 1.481;
   1:  PR[GP1:91,2] = PR[GP1:90,2] + -18.577;
   1:L PR[91] R[100]mm/sec CNT100;
   1:  PR[GP1:91,1] = PR[GP1:90,1] + 6.659;
   1:  PR[GP1:91,2] = PR[GP1:90,2] + -20.667;
   1:L PR[91] R[100]mm/sec CNT100;
   1:  PR[GP1:91,1] = PR[GP1:90,1] + 12.578;
   1:  PR[GP1:91,2] = PR[GP1:90,2] + -21.490;
   1:L PR[91] R[100]mm/sec CNT100;
   1:  PR[GP1:91,1] = PR[GP1:90,1] + 12.657;
   1:  PR[GP1:91,2] = PR[GP1:90,2] + -21.486;
   1:L PR[91] R[100]mm/sec CNT100;
   1:  PR[GP1:91,1] = PR[GP1:90,1] + 18.219;
   1:  PR[GP1:91,2] = PR[GP1:90,2] + -20.838;
   1:L PR[91] R[100]mm/sec CNT100;
   1:  PR[GP1:91,1] = PR[GP1:90,1] + 18.524;
   1:  PR[GP1:91,2] = PR[GP1:90,2] + -20.775;
   1:L PR[91] R[100]mm/sec CNT100;
   1:  PR[GP1:91,1] = PR[GP1:90,1] + 18.918;
   1:  PR[GP1:91,2] = PR[GP1:90,2] + -20.629;
   1:L PR[91] R[100]mm/sec CNT100;
   1:  PR[GP1:91,1] = PR[GP1:90,1] + 23.748;
   1:  PR[GP1:91,2] = PR[GP1:90,2] + -18.751;
   1:L PR[91] R[100]mm/sec CNT100;
   1:  PR[GP1:91,1] = PR[GP1:90,1] + 24.213;
   1:  PR[GP1:91,2] = PR[GP1:90,2] + -18.492;
   1:L PR[91] R[100]mm/sec CNT100;
   1:  PR[GP1:91,1] = PR[GP1:90,1] + 24.779;
   1:  PR[GP1:91,2] = PR[GP1:90,2] + -18.053;
   1:L PR[91] R[100]mm/sec CNT100;
   1:  PR[GP1:91,1] = PR[GP1:90,1] + 28.600;
   1:  PR[GP1:91,2] = PR[GP1:90,2] + -15.278;
   1:L PR[91] R[100]mm/sec CNT100;
   1:  PR[GP1:91,1] = PR[GP1:90,1] + 29.123;
   1:  PR[GP1:91,2] = PR[GP1:90,2] + -14.714;
   1:L PR[91] R[100]mm/sec CNT100;
   1:  PR[GP1:91,1] = PR[GP1:90,1] + 31.804;
   1:  PR[GP1:91,2] = PR[GP1:90,2] + -11.384;
   1:L PR[91] R[100]mm/sec CNT100;
   1:  PR[GP1:91,1] = PR[GP1:90,1] + 32.308;
   1:  PR[GP1:91,2] = PR[GP1:90,2] + -10.623;
   1:L PR[91] R[100]mm/sec CNT100;
   1:  PR[GP1:91,1] = PR[GP1:90,1] + 34.325;
   1:  PR[GP1:91,2] = PR[GP1:90,2] + -6.078;
   1:L PR[91] R[100]mm/sec CNT100;
   1:  PR[GP1:91,1] = PR[GP1:90,1] + 34.556;
   1:  PR[GP1:91,2] = PR[GP1:90,2] + -5.199;
   1:L PR[91] R[100]mm/sec CNT100;
   1:  PR[GP1:91,1] = PR[GP1:90,1] + 34.649;
   1:  PR[GP1:91,2] = PR[GP1:90,2] + -4.066;
   1:L PR[91] R[100]mm/sec CNT100;
   1:  PR[GP1:91,1] = PR[GP1:90,1] + 35.174;
   1:  PR[GP1:91,2] = PR[GP1:90,2] + -0.271;
   1:L PR[91] R[100]mm/sec CNT100;
   1:  PR[GP1:91,1] = PR[GP1:90,1] + 35.088;
   1:  PR[GP1:91,2] = PR[GP1:90,2] + 0.783;
   1:L PR[91] R[100]mm/sec CNT100;
   1:  PR[GP1:91,1] = PR[GP1:90,1] + 34.567;
   1:  PR[GP1:91,2] = PR[GP1:90,2] + 4.531;
   1:L PR[91] R[100]mm/sec CNT100;
   1:  PR[GP1:91,1] = PR[GP1:90,1] + 34.328;
   1:  PR[GP1:91,2] = PR[GP1:90,2] + 5.443;
   1:L PR[91] R[100]mm/sec CNT100;
   1:  PR[GP1:91,1] = PR[GP1:90,1] + 33.889;
   1:  PR[GP1:91,2] = PR[GP1:90,2] + 6.408;
   1:L PR[91] R[100]mm/sec CNT100;
   1:  PR[GP1:91,1] = PR[GP1:90,1] + 32.312;
   1:  PR[GP1:91,2] = PR[GP1:90,2] + 9.992;
   1:L PR[91] R[100]mm/sec CNT100;
   1:  PR[GP1:91,1] = PR[GP1:90,1] + 31.809;
   1:  PR[GP1:91,2] = PR[GP1:90,2] + 10.751;
   1:L PR[91] R[100]mm/sec CNT100;
   1:  PR[GP1:91,1] = PR[GP1:90,1] + 29.135;
   1:  PR[GP1:91,2] = PR[GP1:90,2] + 14.079;
   1:L PR[91] R[100]mm/sec CNT100;
   1:  PR[GP1:91,1] = PR[GP1:90,1] + 28.596;
   1:  PR[GP1:91,2] = PR[GP1:90,2] + 14.660;
   1:L PR[91] R[100]mm/sec CNT100;
   1:  PR[GP1:91,1] = PR[GP1:90,1] + 28.008;
   1:  PR[GP1:91,2] = PR[GP1:90,2] + 15.118;
   1:L PR[91] R[100]mm/sec CNT100;
   1:  PR[GP1:91,1] = PR[GP1:90,1] + 24.255;
   1:  PR[GP1:91,2] = PR[GP1:90,2] + 17.845;
   1:L PR[91] R[100]mm/sec CNT100;
   1:  PR[GP1:91,1] = PR[GP1:90,1] + 23.781;
   1:  PR[GP1:91,2] = PR[GP1:90,2] + 18.109;
   1:L PR[91] R[100]mm/sec CNT100;
   1:  PR[GP1:91,1] = PR[GP1:90,1] + 23.243;
   1:  PR[GP1:91,2] = PR[GP1:90,2] + 18.306;
   1:L PR[91] R[100]mm/sec CNT100;
   1:  PR[GP1:91,1] = PR[GP1:90,1] + 18.543;
   1:  PR[GP1:91,2] = PR[GP1:90,2] + 20.145;
   1:L PR[91] R[100]mm/sec CNT100;
   1:  PR[GP1:91,1] = PR[GP1:90,1] + 18.250;
   1:  PR[GP1:91,2] = PR[GP1:90,2] + 20.206;
   1:L PR[91] R[100]mm/sec CNT100;
   1:  PR[GP1:91,1] = PR[GP1:90,1] + 12.701;
   1:  PR[GP1:91,2] = PR[GP1:90,2] + 20.862;
   1:L PR[91] R[100]mm/sec CNT100;
   1:  PR[GP1:91,1] = PR[GP1:90,1] + 12.594;
   1:  PR[GP1:91,2] = PR[GP1:90,2] + 20.868;
   1:L PR[91] R[100]mm/sec CNT100;
   1:  PR[GP1:91,1] = PR[GP1:90,1] + 12.496;
   1:  PR[GP1:91,2] = PR[GP1:90,2] + 20.858;
   1:L PR[91] R[100]mm/sec CNT100;
   1:  PR[GP1:91,1] = PR[GP1:90,1] + 6.690;
   1:  PR[GP1:91,2] = PR[GP1:90,2] + 20.052;
   1:L PR[91] R[100]mm/sec CNT100;
   1:  PR[GP1:91,1] = PR[GP1:90,1] + 1.268;
   1:  PR[GP1:91,2] = PR[GP1:90,2] + 17.886;
   1:L PR[91] R[100]mm/sec CNT100;
   1:  PR[GP1:91,1] = PR[GP1:90,1] + 0.302;
   1:  PR[GP1:91,2] = PR[GP1:90,2] + 17.476;
   1:L PR[91] R[100]mm/sec CNT100;
   1:  PR[91] = PR[90];
   1:  PR[GP1:91,1] = PR[GP1:90,1] + -0.823;
   1:  PR[GP1:91,2] = PR[GP1:90,2] + 18.037;
   1:  PR[GP1:91,3] = PR[GP1:90,3] + 41.785;
   1:L PR[91] R[100]mm/sec CNT100;
   1:  PR[GP1:91,1] = PR[GP1:90,1] + -1.082;
   1:  PR[GP1:91,2] = PR[GP1:90,2] + 18.075;
   1:L PR[91] R[100]mm/sec CNT100;
   1:  PR[GP1:91,1] = PR[GP1:90,1] + -6.160;
   1:  PR[GP1:91,2] = PR[GP1:90,2] + 20.103;
   1:L PR[91] R[100]mm/sec CNT100;
   1:  PR[GP1:91,1] = PR[GP1:90,1] + -6.289;
   1:  PR[GP1:91,2] = PR[GP1:90,2] + 20.149;
   1:L PR[91] R[100]mm/sec CNT100;
   1:  PR[GP1:91,1] = PR[GP1:90,1] + -9.227;
   1:  PR[GP1:91,2] = PR[GP1:90,2] + 20.518;
   1:L PR[91] R[100]mm/sec CNT100;
   1:  PR[GP1:91,1] = PR[GP1:90,1] + -12.197;
   1:  PR[GP1:91,2] = PR[GP1:90,2] + 20.924;
   1:L PR[91] R[100]mm/sec CNT100;
   1:  PR[GP1:91,1] = PR[GP1:90,1] + -17.975;
   1:  PR[GP1:91,2] = PR[GP1:90,2] + 20.248;
   1:L PR[91] R[100]mm/sec CNT100;
   1:  PR[GP1:91,1] = PR[GP1:90,1] + -18.147;
   1:  PR[GP1:91,2] = PR[GP1:90,2] + 20.212;
   1:L PR[91] R[100]mm/sec CNT100;
   1:  PR[GP1:91,1] = PR[GP1:90,1] + -18.399;
   1:  PR[GP1:91,2] = PR[GP1:90,2] + 20.119;
   1:L PR[91] R[100]mm/sec CNT100;
   1:  PR[GP1:91,1] = PR[GP1:90,1] + -23.455;
   1:  PR[GP1:91,2] = PR[GP1:90,2] + 18.143;
   1:L PR[91] R[100]mm/sec CNT100;
   1:  PR[GP1:91,1] = PR[GP1:90,1] + -23.797;
   1:  PR[GP1:91,2] = PR[GP1:90,2] + 17.951;
   1:L PR[91] R[100]mm/sec CNT100;
   1:  PR[GP1:91,1] = PR[GP1:90,1] + -24.245;
   1:  PR[GP1:91,2] = PR[GP1:90,2] + 17.602;
   1:L PR[91] R[100]mm/sec CNT100;
   1:  PR[GP1:91,1] = PR[GP1:90,1] + -28.273;
   1:  PR[GP1:91,2] = PR[GP1:90,2] + 14.668;
   1:L PR[91] R[100]mm/sec CNT100;
   1:  PR[GP1:91,1] = PR[GP1:90,1] + -28.695;
   1:  PR[GP1:91,2] = PR[GP1:90,2] + 14.212;
   1:L PR[91] R[100]mm/sec CNT100;
   1:  PR[GP1:91,1] = PR[GP1:90,1] + -31.529;
   1:  PR[GP1:91,2] = PR[GP1:90,2] + 10.694;
   1:L PR[91] R[100]mm/sec CNT100;
   1:  PR[GP1:91,1] = PR[GP1:90,1] + -31.945;
   1:  PR[GP1:91,2] = PR[GP1:90,2] + 10.061;
   1:L PR[91] R[100]mm/sec CNT100;
   1:  PR[GP1:91,1] = PR[GP1:90,1] + -33.999;
   1:  PR[GP1:91,2] = PR[GP1:90,2] + 5.394;
   1:L PR[91] R[100]mm/sec CNT100;
   1:  PR[GP1:91,1] = PR[GP1:90,1] + -34.195;
   1:  PR[GP1:91,2] = PR[GP1:90,2] + 4.638;
   1:L PR[91] R[100]mm/sec CNT100;
   1:  PR[GP1:91,1] = PR[GP1:90,1] + -34.271;
   1:  PR[GP1:91,2] = PR[GP1:90,2] + 3.683;
   1:L PR[91] R[100]mm/sec CNT100;
   1:  PR[GP1:91,1] = PR[GP1:90,1] + -34.831;
   1:  PR[GP1:91,2] = PR[GP1:90,2] + -0.354;
   1:L PR[91] R[100]mm/sec CNT100;
   1:  PR[GP1:91,1] = PR[GP1:90,1] + -34.761;
   1:  PR[GP1:91,2] = PR[GP1:90,2] + -1.232;
   1:L PR[91] R[100]mm/sec CNT100;
   1:  PR[GP1:91,1] = PR[GP1:90,1] + -34.204;
   1:  PR[GP1:91,2] = PR[GP1:90,2] + -5.226;
   1:L PR[91] R[100]mm/sec CNT100;
   1:  PR[GP1:91,1] = PR[GP1:90,1] + -33.999;
   1:  PR[GP1:91,2] = PR[GP1:90,2] + -6.018;
   1:L PR[91] R[100]mm/sec CNT100;
   1:  PR[GP1:91,1] = PR[GP1:90,1] + -33.619;
   1:  PR[GP1:91,2] = PR[GP1:90,2] + -6.866;
   1:L PR[91] R[100]mm/sec CNT100;
   1:  PR[GP1:91,1] = PR[GP1:90,1] + -31.939;
   1:  PR[GP1:91,2] = PR[GP1:90,2] + -10.695;
   1:L PR[91] R[100]mm/sec CNT100;
   1:  PR[GP1:91,1] = PR[GP1:90,1] + -31.523;
   1:  PR[GP1:91,2] = PR[GP1:90,2] + -11.327;
   1:L PR[91] R[100]mm/sec CNT100;
   1:  PR[GP1:91,1] = PR[GP1:90,1] + -28.682;
   1:  PR[GP1:91,2] = PR[GP1:90,2] + -14.849;
   1:L PR[91] R[100]mm/sec CNT100;
   1:  PR[GP1:91,1] = PR[GP1:90,1] + -28.242;
   1:  PR[GP1:91,2] = PR[GP1:90,2] + -15.323;
   1:L PR[91] R[100]mm/sec CNT100;
   1:  PR[GP1:91,1] = PR[GP1:90,1] + -27.758;
   1:  PR[GP1:91,2] = PR[GP1:90,2] + -15.702;
   1:L PR[91] R[100]mm/sec CNT100;
   1:  PR[GP1:91,1] = PR[GP1:90,1] + -23.795;
   1:  PR[GP1:91,2] = PR[GP1:90,2] + -18.576;
   1:L PR[91] R[100]mm/sec CNT100;
   1:  PR[GP1:91,1] = PR[GP1:90,1] + -23.433;
   1:  PR[GP1:91,2] = PR[GP1:90,2] + -18.778;
   1:L PR[91] R[100]mm/sec CNT100;
   1:  PR[GP1:91,1] = PR[GP1:90,1] + -18.101;
   1:  PR[GP1:91,2] = PR[GP1:90,2] + -20.847;
   1:L PR[91] R[100]mm/sec CNT100;
   1:  PR[GP1:91,1] = PR[GP1:90,1] + -17.941;
   1:  PR[GP1:91,2] = PR[GP1:90,2] + -20.881;
   1:L PR[91] R[100]mm/sec CNT100;
   1:  PR[GP1:91,1] = PR[GP1:90,1] + -12.187;
   1:  PR[GP1:91,2] = PR[GP1:90,2] + -21.551;
   1:L PR[91] R[100]mm/sec CNT100;
   1:  PR[GP1:91,1] = PR[GP1:90,1] + -12.143;
   1:  PR[GP1:91,2] = PR[GP1:90,2] + -21.550;
   1:L PR[91] R[100]mm/sec CNT100;
   1:  PR[GP1:91,1] = PR[GP1:90,1] + -9.233;
   1:  PR[GP1:91,2] = PR[GP1:90,2] + -21.143;
   1:L PR[91] R[100]mm/sec CNT100;
   1:  PR[GP1:91,1] = PR[GP1:90,1] + -6.254;
   1:  PR[GP1:91,2] = PR[GP1:90,2] + -20.762;
   1:L PR[91] R[100]mm/sec CNT100;
   1:  PR[GP1:91,1] = PR[GP1:90,1] + -5.298;
   1:  PR[GP1:91,2] = PR[GP1:90,2] + -20.394;
   1:L PR[91] R[100]mm/sec CNT100;
   1:  PR[GP1:91,1] = PR[GP1:90,1] + -1.101;
   1:  PR[GP1:91,2] = PR[GP1:90,2] + -18.702;
   1:L PR[91] R[100]mm/sec CNT100;
   1:  PR[GP1:91,1] = PR[GP1:90,1] + -0.529;
   1:  PR[GP1:91,2] = PR[GP1:90,2] + -18.605;
   1:L PR[91] R[100]mm/sec CNT100;
   1:  PR[GP1:91,1] = PR[GP1:90,1] + -0.441;
   1:  PR[GP1:91,2] = PR[GP1:90,2] + -18.579;
   1:L PR[91] R[100]mm/sec CNT100;
   1:  PR[GP1:91,1] = PR[GP1:90,1] + 0.157;
   1:  PR[GP1:91,2] = PR[GP1:90,2] + -18.332;
   1:L PR[91] R[100]mm/sec CNT100;
   1:  PR[GP1:91,1] = PR[GP1:90,1] + 1.218;
   1:  PR[GP1:91,2] = PR[GP1:90,2] + -18.658;
   1:L PR[91] R[100]mm/sec CNT100;
   1:  PR[GP1:91,1] = PR[GP1:90,1] + 1.464;
   1:  PR[GP1:91,2] = PR[GP1:90,2] + -18.786;
   1:L PR[91] R[100]mm/sec CNT100;
   1:  PR[GP1:91,1] = PR[GP1:90,1] + 5.452;
   1:  PR[GP1:91,2] = PR[GP1:90,2] + -20.392;
   1:L PR[91] R[100]mm/sec CNT100;
   1:  PR[GP1:91,1] = PR[GP1:90,1] + 6.389;
   1:  PR[GP1:91,2] = PR[GP1:90,2] + -20.754;
   1:L PR[91] R[100]mm/sec CNT100;
   1:  PR[GP1:91,1] = PR[GP1:90,1] + 9.387;
   1:  PR[GP1:91,2] = PR[GP1:90,2] + -21.142;
   1:L PR[91] R[100]mm/sec CNT100;
   1:  PR[GP1:91,1] = PR[GP1:90,1] + 12.306;
   1:  PR[GP1:91,2] = PR[GP1:90,2] + -21.548;
   1:L PR[91] R[100]mm/sec CNT100;
   1:  PR[GP1:91,1] = PR[GP1:90,1] + 18.094;
   1:  PR[GP1:91,2] = PR[GP1:90,2] + -20.881;
   1:L PR[91] R[100]mm/sec CNT100;
   1:  PR[GP1:91,1] = PR[GP1:90,1] + 18.265;
   1:  PR[GP1:91,2] = PR[GP1:90,2] + -20.845;
   1:L PR[91] R[100]mm/sec CNT100;
   1:  PR[GP1:91,1] = PR[GP1:90,1] + 18.517;
   1:  PR[GP1:91,2] = PR[GP1:90,2] + -20.752;
   1:L PR[91] R[100]mm/sec CNT100;
   1:  PR[GP1:91,1] = PR[GP1:90,1] + 23.586;
   1:  PR[GP1:91,2] = PR[GP1:90,2] + -18.781;
   1:L PR[91] R[100]mm/sec CNT100;
   1:  PR[GP1:91,1] = PR[GP1:90,1] + 23.926;
   1:  PR[GP1:91,2] = PR[GP1:90,2] + -18.592;
   1:L PR[91] R[100]mm/sec CNT100;
   1:  PR[GP1:91,1] = PR[GP1:90,1] + 24.368;
   1:  PR[GP1:91,2] = PR[GP1:90,2] + -18.249;
   1:L PR[91] R[100]mm/sec CNT100;
   1:  PR[GP1:91,1] = PR[GP1:90,1] + 28.405;
   1:  PR[GP1:91,2] = PR[GP1:90,2] + -15.316;
   1:L PR[91] R[100]mm/sec CNT100;
   1:  PR[GP1:91,1] = PR[GP1:90,1] + 28.828;
   1:  PR[GP1:91,2] = PR[GP1:90,2] + -14.861;
   1:L PR[91] R[100]mm/sec CNT100;
   1:  PR[GP1:91,1] = PR[GP1:90,1] + 31.670;
   1:  PR[GP1:91,2] = PR[GP1:90,2] + -11.331;
   1:L PR[91] R[100]mm/sec CNT100;
   1:  PR[GP1:91,1] = PR[GP1:90,1] + 32.093;
   1:  PR[GP1:91,2] = PR[GP1:90,2] + -10.692;
   1:L PR[91] R[100]mm/sec CNT100;
   1:  PR[GP1:91,1] = PR[GP1:90,1] + 34.151;
   1:  PR[GP1:91,2] = PR[GP1:90,2] + -6.051;
   1:L PR[91] R[100]mm/sec CNT100;
   1:  PR[GP1:91,1] = PR[GP1:90,1] + 34.346;
   1:  PR[GP1:91,2] = PR[GP1:90,2] + -5.306;
   1:L PR[91] R[100]mm/sec CNT100;
   1:  PR[GP1:91,1] = PR[GP1:90,1] + 34.427;
   1:  PR[GP1:91,2] = PR[GP1:90,2] + -4.322;
   1:L PR[91] R[100]mm/sec CNT100;
   1:  PR[GP1:91,1] = PR[GP1:90,1] + 34.988;
   1:  PR[GP1:91,2] = PR[GP1:90,2] + -0.271;
   1:L PR[91] R[100]mm/sec CNT100;
   1:  PR[GP1:91,1] = PR[GP1:90,1] + 34.913;
   1:  PR[GP1:91,2] = PR[GP1:90,2] + 0.639;
   1:L PR[91] R[100]mm/sec CNT100;
   1:  PR[GP1:91,1] = PR[GP1:90,1] + 34.358;
   1:  PR[GP1:91,2] = PR[GP1:90,2] + 4.638;
   1:L PR[91] R[100]mm/sec CNT100;
   1:  PR[GP1:91,1] = PR[GP1:90,1] + 34.154;
   1:  PR[GP1:91,2] = PR[GP1:90,2] + 5.416;
   1:L PR[91] R[100]mm/sec CNT100;
   1:  PR[GP1:91,1] = PR[GP1:90,1] + 33.774;
   1:  PR[GP1:91,2] = PR[GP1:90,2] + 6.251;
   1:L PR[91] R[100]mm/sec CNT100;
   1:  PR[GP1:91,1] = PR[GP1:90,1] + 32.098;
   1:  PR[GP1:91,2] = PR[GP1:90,2] + 10.060;
   1:L PR[91] R[100]mm/sec CNT100;
   1:  PR[GP1:91,1] = PR[GP1:90,1] + 31.675;
   1:  PR[GP1:91,2] = PR[GP1:90,2] + 10.698;
   1:L PR[91] R[100]mm/sec CNT100;
   1:  PR[GP1:91,1] = PR[GP1:90,1] + 28.840;
   1:  PR[GP1:91,2] = PR[GP1:90,2] + 14.225;
   1:L PR[91] R[100]mm/sec CNT100;
   1:  PR[GP1:91,1] = PR[GP1:90,1] + 28.402;
   1:  PR[GP1:91,2] = PR[GP1:90,2] + 14.698;
   1:L PR[91] R[100]mm/sec CNT100;
   1:  PR[GP1:91,1] = PR[GP1:90,1] + 27.921;
   1:  PR[GP1:91,2] = PR[GP1:90,2] + 15.073;
   1:L PR[91] R[100]mm/sec CNT100;
   1:  PR[GP1:91,1] = PR[GP1:90,1] + 23.969;
   1:  PR[GP1:91,2] = PR[GP1:90,2] + 17.944;
   1:L PR[91] R[100]mm/sec CNT100;
   1:  PR[GP1:91,1] = PR[GP1:90,1] + 23.621;
   1:  PR[GP1:91,2] = PR[GP1:90,2] + 18.138;
   1:L PR[91] R[100]mm/sec CNT100;
   1:  PR[GP1:91,1] = PR[GP1:90,1] + 23.205;
   1:  PR[GP1:91,2] = PR[GP1:90,2] + 18.291;
   1:L PR[91] R[100]mm/sec CNT100;
   1:  PR[GP1:91,1] = PR[GP1:90,1] + 18.286;
   1:  PR[GP1:91,2] = PR[GP1:90,2] + 20.215;
   1:L PR[91] R[100]mm/sec CNT100;
   1:  PR[GP1:91,1] = PR[GP1:90,1] + 18.125;
   1:  PR[GP1:91,2] = PR[GP1:90,2] + 20.249;
   1:L PR[91] R[100]mm/sec CNT100;
   1:  PR[GP1:91,1] = PR[GP1:90,1] + 12.386;
   1:  PR[GP1:91,2] = PR[GP1:90,2] + 20.927;
   1:L PR[91] R[100]mm/sec CNT100;
   1:  PR[GP1:91,1] = PR[GP1:90,1] + 12.341;
   1:  PR[GP1:91,2] = PR[GP1:90,2] + 20.926;
   1:L PR[91] R[100]mm/sec CNT100;
   1:  PR[GP1:91,1] = PR[GP1:90,1] + 9.385;
   1:  PR[GP1:91,2] = PR[GP1:90,2] + 20.518;
   1:L PR[91] R[100]mm/sec CNT100;
   1:  PR[GP1:91,1] = PR[GP1:90,1] + 6.442;
   1:  PR[GP1:91,2] = PR[GP1:90,2] + 20.147;
   1:L PR[91] R[100]mm/sec CNT100;
   1:  PR[GP1:91,1] = PR[GP1:90,1] + 6.312;
   1:  PR[GP1:91,2] = PR[GP1:90,2] + 20.100;
   1:L PR[91] R[100]mm/sec CNT100;
   1:  PR[GP1:91,1] = PR[GP1:90,1] + 1.340;
   1:  PR[GP1:91,2] = PR[GP1:90,2] + 18.117;
   1:L PR[91] R[100]mm/sec CNT100;
   1:  PR[GP1:91,1] = PR[GP1:90,1] + 1.100;
   1:  PR[GP1:91,2] = PR[GP1:90,2] + 18.042;
   1:L PR[91] R[100]mm/sec CNT100;
   1:  PR[GP1:91,1] = PR[GP1:90,1] + 0.322;
   1:  PR[GP1:91,2] = PR[GP1:90,2] + 17.713;
   1:L PR[91] R[100]mm/sec CNT100;
   1:  PR[91] = PR[90];
   1:  PR[GP1:91,1] = PR[GP1:90,1] + -0.534;
   1:  PR[GP1:91,2] = PR[GP1:90,2] + 18.197;
   1:  PR[GP1:91,3] = PR[GP1:90,3] + 42.395;
   1:L PR[91] R[100]mm/sec CNT100;
   1:  PR[GP1:91,1] = PR[GP1:90,1] + -1.065;
   1:  PR[GP1:91,2] = PR[GP1:90,2] + 18.274;
   1:L PR[91] R[100]mm/sec CNT100;
   1:  PR[GP1:91,1] = PR[GP1:90,1] + -5.585;
   1:  PR[GP1:91,2] = PR[GP1:90,2] + 20.080;
   1:L PR[91] R[100]mm/sec CNT100;
   1:  PR[GP1:91,1] = PR[GP1:90,1] + -6.072;
   1:  PR[GP1:91,2] = PR[GP1:90,2] + 20.254;
   1:L PR[91] R[100]mm/sec CNT100;
   1:  PR[GP1:91,1] = PR[GP1:90,1] + -11.929;
   1:  PR[GP1:91,2] = PR[GP1:90,2] + 20.990;
   1:L PR[91] R[100]mm/sec CNT100;
   1:  PR[GP1:91,1] = PR[GP1:90,1] + -17.849;
   1:  PR[GP1:91,2] = PR[GP1:90,2] + 20.291;
   1:L PR[91] R[100]mm/sec CNT100;
   1:  PR[GP1:91,1] = PR[GP1:90,1] + -17.889;
   1:  PR[GP1:91,2] = PR[GP1:90,2] + 20.283;
   1:L PR[91] R[100]mm/sec CNT100;
   1:  PR[GP1:91,1] = PR[GP1:90,1] + -17.998;
   1:  PR[GP1:91,2] = PR[GP1:90,2] + 20.243;
   1:L PR[91] R[100]mm/sec CNT100;
   1:  PR[GP1:91,1] = PR[GP1:90,1] + -23.293;
   1:  PR[GP1:91,2] = PR[GP1:90,2] + 18.172;
   1:L PR[91] R[100]mm/sec CNT100;
   1:  PR[GP1:91,1] = PR[GP1:90,1] + -23.509;
   1:  PR[GP1:91,2] = PR[GP1:90,2] + 18.051;
   1:L PR[91] R[100]mm/sec CNT100;
   1:  PR[GP1:91,1] = PR[GP1:90,1] + -23.833;
   1:  PR[GP1:91,2] = PR[GP1:90,2] + 17.799;
   1:L PR[91] R[100]mm/sec CNT100;
   1:  PR[GP1:91,1] = PR[GP1:90,1] + -28.077;
   1:  PR[GP1:91,2] = PR[GP1:90,2] + 14.709;
   1:L PR[91] R[100]mm/sec CNT100;
   1:  PR[GP1:91,1] = PR[GP1:90,1] + -28.399;
   1:  PR[GP1:91,2] = PR[GP1:90,2] + 14.360;
   1:L PR[91] R[100]mm/sec CNT100;
   1:  PR[GP1:91,1] = PR[GP1:90,1] + -31.393;
   1:  PR[GP1:91,2] = PR[GP1:90,2] + 10.643;
   1:L PR[91] R[100]mm/sec CNT100;
   1:  PR[GP1:91,1] = PR[GP1:90,1] + -31.730;
   1:  PR[GP1:91,2] = PR[GP1:90,2] + 10.130;
   1:L PR[91] R[100]mm/sec CNT100;
   1:  PR[GP1:91,1] = PR[GP1:90,1] + -33.824;
   1:  PR[GP1:91,2] = PR[GP1:90,2] + 5.369;
   1:L PR[91] R[100]mm/sec CNT100;
   1:  PR[GP1:91,1] = PR[GP1:90,1] + -33.985;
   1:  PR[GP1:91,2] = PR[GP1:90,2] + 4.750;
   1:L PR[91] R[100]mm/sec CNT100;
   1:  PR[GP1:91,1] = PR[GP1:90,1] + -34.050;
   1:  PR[GP1:91,2] = PR[GP1:90,2] + 3.938;
   1:L PR[91] R[100]mm/sec CNT100;
   1:  PR[GP1:91,1] = PR[GP1:90,1] + -34.645;
   1:  PR[GP1:91,2] = PR[GP1:90,2] + -0.354;
   1:L PR[91] R[100]mm/sec CNT100;
   1:  PR[GP1:91,1] = PR[GP1:90,1] + -34.586;
   1:  PR[GP1:91,2] = PR[GP1:90,2] + -1.093;
   1:L PR[91] R[100]mm/sec CNT100;
   1:  PR[GP1:91,1] = PR[GP1:90,1] + -33.994;
   1:  PR[GP1:91,2] = PR[GP1:90,2] + -5.338;
   1:L PR[91] R[100]mm/sec CNT100;
   1:  PR[GP1:91,1] = PR[GP1:90,1] + -33.824;
   1:  PR[GP1:91,2] = PR[GP1:90,2] + -5.993;
   1:L PR[91] R[100]mm/sec CNT100;
   1:  PR[GP1:91,1] = PR[GP1:90,1] + -33.503;
   1:  PR[GP1:91,2] = PR[GP1:90,2] + -6.709;
   1:L PR[91] R[100]mm/sec CNT100;
   1:  PR[GP1:91,1] = PR[GP1:90,1] + -31.724;
   1:  PR[GP1:91,2] = PR[GP1:90,2] + -10.765;
   1:L PR[91] R[100]mm/sec CNT100;
   1:  PR[GP1:91,1] = PR[GP1:90,1] + -31.387;
   1:  PR[GP1:91,2] = PR[GP1:90,2] + -11.276;
   1:L PR[91] R[100]mm/sec CNT100;
   1:  PR[GP1:91,1] = PR[GP1:90,1] + -28.385;
   1:  PR[GP1:91,2] = PR[GP1:90,2] + -14.998;
   1:L PR[91] R[100]mm/sec CNT100;
   1:  PR[GP1:91,1] = PR[GP1:90,1] + -28.046;
   1:  PR[GP1:91,2] = PR[GP1:90,2] + -15.364;
   1:L PR[91] R[100]mm/sec CNT100;
   1:  PR[GP1:91,1] = PR[GP1:90,1] + -27.669;
   1:  PR[GP1:91,2] = PR[GP1:90,2] + -15.659;
   1:L PR[91] R[100]mm/sec CNT100;
   1:  PR[GP1:91,1] = PR[GP1:90,1] + -23.506;
   1:  PR[GP1:91,2] = PR[GP1:90,2] + -18.677;
   1:L PR[91] R[100]mm/sec CNT100;
   1:  PR[GP1:91,1] = PR[GP1:90,1] + -23.270;
   1:  PR[GP1:91,2] = PR[GP1:90,2] + -18.809;
   1:L PR[91] R[100]mm/sec CNT100;
   1:  PR[GP1:91,1] = PR[GP1:90,1] + -17.841;
   1:  PR[GP1:91,2] = PR[GP1:90,2] + -20.919;
   1:L PR[91] R[100]mm/sec CNT100;
   1:  PR[GP1:91,1] = PR[GP1:90,1] + -17.814;
   1:  PR[GP1:91,2] = PR[GP1:90,2] + -20.924;
   1:L PR[91] R[100]mm/sec CNT100;
   1:  PR[GP1:91,1] = PR[GP1:90,1] + -11.881;
   1:  PR[GP1:91,2] = PR[GP1:90,2] + -21.614;
   1:L PR[91] R[100]mm/sec CNT100;
   1:  PR[GP1:91,1] = PR[GP1:90,1] + -6.014;
   1:  PR[GP1:91,2] = PR[GP1:90,2] + -20.864;
   1:L PR[91] R[100]mm/sec CNT100;
   1:  PR[GP1:91,1] = PR[GP1:90,1] + -5.777;
   1:  PR[GP1:91,2] = PR[GP1:90,2] + -20.781;
   1:L PR[91] R[100]mm/sec CNT100;
   1:  PR[GP1:91,1] = PR[GP1:90,1] + -3.769;
   1:  PR[GP1:91,2] = PR[GP1:90,2] + -19.994;
   1:L PR[91] R[100]mm/sec CNT100;
   1:  PR[GP1:91,1] = PR[GP1:90,1] + -1.084;
   1:  PR[GP1:91,2] = PR[GP1:90,2] + -18.912;
   1:L PR[91] R[100]mm/sec CNT100;
   1:  PR[GP1:91,1] = PR[GP1:90,1] + -0.388;
   1:  PR[GP1:91,2] = PR[GP1:90,2] + -18.793;
   1:L PR[91] R[100]mm/sec CNT100;
   1:  PR[GP1:91,1] = PR[GP1:90,1] + 0.221;
   1:  PR[GP1:91,2] = PR[GP1:90,2] + -18.582;
   1:L PR[91] R[100]mm/sec CNT100;
   1:  PR[GP1:91,1] = PR[GP1:90,1] + 1.273;
   1:  PR[GP1:91,2] = PR[GP1:90,2] + -18.905;
   1:L PR[91] R[100]mm/sec CNT100;
   1:  PR[GP1:91,1] = PR[GP1:90,1] + 1.447;
   1:  PR[GP1:91,2] = PR[GP1:90,2] + -18.996;
   1:L PR[91] R[100]mm/sec CNT100;
   1:  PR[GP1:91,1] = PR[GP1:90,1] + 3.922;
   1:  PR[GP1:91,2] = PR[GP1:90,2] + -19.992;
   1:L PR[91] R[100]mm/sec CNT100;
   1:  PR[GP1:91,1] = PR[GP1:90,1] + 5.933;
   1:  PR[GP1:91,2] = PR[GP1:90,2] + -20.780;
   1:L PR[91] R[100]mm/sec CNT100;
   1:  PR[GP1:91,1] = PR[GP1:90,1] + 6.129;
   1:  PR[GP1:91,2] = PR[GP1:90,2] + -20.849;
   1:L PR[91] R[100]mm/sec CNT100;
   1:  PR[GP1:91,1] = PR[GP1:90,1] + 12.035;
   1:  PR[GP1:91,2] = PR[GP1:90,2] + -21.614;
   1:L PR[91] R[100]mm/sec CNT100;
   1:  PR[GP1:91,1] = PR[GP1:90,1] + 17.968;
   1:  PR[GP1:91,2] = PR[GP1:90,2] + -20.924;
   1:L PR[91] R[100]mm/sec CNT100;
   1:  PR[GP1:91,1] = PR[GP1:90,1] + 18.006;
   1:  PR[GP1:91,2] = PR[GP1:90,2] + -20.916;
   1:L PR[91] R[100]mm/sec CNT100;
   1:  PR[GP1:91,1] = PR[GP1:90,1] + 18.115;
   1:  PR[GP1:91,2] = PR[GP1:90,2] + -20.876;
   1:L PR[91] R[100]mm/sec CNT100;
   1:  PR[GP1:91,1] = PR[GP1:90,1] + 23.424;
   1:  PR[GP1:91,2] = PR[GP1:90,2] + -18.811;
   1:L PR[91] R[100]mm/sec CNT100;
   1:  PR[GP1:91,1] = PR[GP1:90,1] + 23.638;
   1:  PR[GP1:91,2] = PR[GP1:90,2] + -18.692;
   1:L PR[91] R[100]mm/sec CNT100;
   1:  PR[GP1:91,1] = PR[GP1:90,1] + 23.957;
   1:  PR[GP1:91,2] = PR[GP1:90,2] + -18.445;
   1:L PR[91] R[100]mm/sec CNT100;
   1:  PR[GP1:91,1] = PR[GP1:90,1] + 28.210;
   1:  PR[GP1:91,2] = PR[GP1:90,2] + -15.355;
   1:L PR[91] R[100]mm/sec CNT100;
   1:  PR[GP1:91,1] = PR[GP1:90,1] + 28.533;
   1:  PR[GP1:91,2] = PR[GP1:90,2] + -15.008;
   1:L PR[91] R[100]mm/sec CNT100;
   1:  PR[GP1:91,1] = PR[GP1:90,1] + 31.536;
   1:  PR[GP1:91,2] = PR[GP1:90,2] + -11.279;
   1:L PR[91] R[100]mm/sec CNT100;
   1:  PR[GP1:91,1] = PR[GP1:90,1] + 31.878;
   1:  PR[GP1:91,2] = PR[GP1:90,2] + -10.761;
   1:L PR[91] R[100]mm/sec CNT100;
   1:  PR[GP1:91,1] = PR[GP1:90,1] + 33.976;
   1:  PR[GP1:91,2] = PR[GP1:90,2] + -6.024;
   1:L PR[91] R[100]mm/sec CNT100;
   1:  PR[GP1:91,1] = PR[GP1:90,1] + 34.136;
   1:  PR[GP1:91,2] = PR[GP1:90,2] + -5.414;
   1:L PR[91] R[100]mm/sec CNT100;
   1:  PR[GP1:91,1] = PR[GP1:90,1] + 34.205;
   1:  PR[GP1:91,2] = PR[GP1:90,2] + -4.578;
   1:L PR[91] R[100]mm/sec CNT100;
   1:  PR[GP1:91,1] = PR[GP1:90,1] + 34.801;
   1:  PR[GP1:91,2] = PR[GP1:90,2] + -0.271;
   1:L PR[91] R[100]mm/sec CNT100;
   1:  PR[GP1:91,1] = PR[GP1:90,1] + 34.739;
   1:  PR[GP1:91,2] = PR[GP1:90,2] + 0.496;
   1:L PR[91] R[100]mm/sec CNT100;
   1:  PR[GP1:91,1] = PR[GP1:90,1] + 34.148;
   1:  PR[GP1:91,2] = PR[GP1:90,2] + 4.746;
   1:L PR[91] R[100]mm/sec CNT100;
   1:  PR[GP1:91,1] = PR[GP1:90,1] + 33.978;
   1:  PR[GP1:91,2] = PR[GP1:90,2] + 5.395;
   1:L PR[91] R[100]mm/sec CNT100;
   1:  PR[GP1:91,1] = PR[GP1:90,1] + 31.884;
   1:  PR[GP1:91,2] = PR[GP1:90,2] + 10.127;
   1:L PR[91] R[100]mm/sec CNT100;
   1:  PR[GP1:91,1] = PR[GP1:90,1] + 31.541;
   1:  PR[GP1:91,2] = PR[GP1:90,2] + 10.645;
   1:L PR[91] R[100]mm/sec CNT100;
   1:  PR[GP1:91,1] = PR[GP1:90,1] + 28.546;
   1:  PR[GP1:91,2] = PR[GP1:90,2] + 14.371;
   1:L PR[91] R[100]mm/sec CNT100;
   1:  PR[GP1:91,1] = PR[GP1:90,1] + 28.207;
   1:  PR[GP1:91,2] = PR[GP1:90,2] + 14.736;
   1:L PR[91] R[100]mm/sec CNT100;
   1:  PR[GP1:91,1] = PR[GP1:90,1] + 27.834;
   1:  PR[GP1:91,2] = PR[GP1:90,2] + 15.027;
   1:L PR[91] R[100]mm/sec CNT100;
   1:  PR[GP1:91,1] = PR[GP1:90,1] + 23.682;
   1:  PR[GP1:91,2] = PR[GP1:90,2] + 18.044;
   1:L PR[91] R[100]mm/sec CNT100;
   1:  PR[GP1:91,1] = PR[GP1:90,1] + 23.448;
   1:  PR[GP1:91,2] = PR[GP1:90,2] + 18.175;
   1:L PR[91] R[100]mm/sec CNT100;
   1:  PR[GP1:91,1] = PR[GP1:90,1] + 18.030;
   1:  PR[GP1:91,2] = PR[GP1:90,2] + 20.286;
   1:L PR[91] R[100]mm/sec CNT100;
   1:  PR[GP1:91,1] = PR[GP1:90,1] + 18.001;
   1:  PR[GP1:91,2] = PR[GP1:90,2] + 20.291;
   1:L PR[91] R[100]mm/sec CNT100;
   1:  PR[GP1:91,1] = PR[GP1:90,1] + 12.082;
   1:  PR[GP1:91,2] = PR[GP1:90,2] + 20.990;
   1:L PR[91] R[100]mm/sec CNT100;
   1:  PR[GP1:91,1] = PR[GP1:90,1] + 6.225;
   1:  PR[GP1:91,2] = PR[GP1:90,2] + 20.252;
   1:L PR[91] R[100]mm/sec CNT100;
   1:  PR[GP1:91,1] = PR[GP1:90,1] + 5.737;
   1:  PR[GP1:91,2] = PR[GP1:90,2] + 20.077;
   1:L PR[91] R[100]mm/sec CNT100;
   1:  PR[GP1:91,1] = PR[GP1:90,1] + 1.291;
   1:  PR[GP1:91,2] = PR[GP1:90,2] + 18.303;
   1:L PR[91] R[100]mm/sec CNT100;
   1:  PR[GP1:91,1] = PR[GP1:90,1] + 1.036;
   1:  PR[GP1:91,2] = PR[GP1:90,2] + 18.237;
   1:L PR[91] R[100]mm/sec CNT100;
   1:  PR[GP1:91,1] = PR[GP1:90,1] + 0.328;
   1:  PR[GP1:91,2] = PR[GP1:90,2] + 17.953;
   1:L PR[91] R[100]mm/sec CNT100;
   1:  PR[91] = PR[90];
   1:  PR[GP1:91,1] = PR[GP1:90,1] + -0.245;
   1:  PR[GP1:91,2] = PR[GP1:90,2] + 18.357;
   1:  PR[GP1:91,3] = PR[GP1:90,3] + 43.005;
   1:L PR[91] R[100]mm/sec CNT100;
   1:  PR[GP1:91,1] = PR[GP1:90,1] + -1.048;
   1:  PR[GP1:91,2] = PR[GP1:90,2] + 18.474;
   1:L PR[91] R[100]mm/sec CNT100;
   1:  PR[GP1:91,1] = PR[GP1:90,1] + -5.009;
   1:  PR[GP1:91,2] = PR[GP1:90,2] + 20.056;
   1:L PR[91] R[100]mm/sec CNT100;
   1:  PR[GP1:91,1] = PR[GP1:90,1] + -5.856;
   1:  PR[GP1:91,2] = PR[GP1:90,2] + 20.359;
   1:L PR[91] R[100]mm/sec CNT100;
   1:  PR[GP1:91,1] = PR[GP1:90,1] + -11.620;
   1:  PR[GP1:91,2] = PR[GP1:90,2] + 21.083;
   1:L PR[91] R[100]mm/sec CNT100;
   1:  PR[GP1:91,1] = PR[GP1:90,1] + -11.738;
   1:  PR[GP1:91,2] = PR[GP1:90,2] + 21.095;
   1:L PR[91] R[100]mm/sec CNT100;
   1:  PR[GP1:91,1] = PR[GP1:90,1] + -15.768;
   1:  PR[GP1:91,2] = PR[GP1:90,2] + 20.566;
   1:L PR[91] R[100]mm/sec CNT100;
   1:  PR[GP1:91,1] = PR[GP1:90,1] + -17.659;
   1:  PR[GP1:91,2] = PR[GP1:90,2] + 20.342;
   1:L PR[91] R[100]mm/sec CNT100;
   1:  PR[GP1:91,1] = PR[GP1:90,1] + -23.132;
   1:  PR[GP1:91,2] = PR[GP1:90,2] + 18.202;
   1:L PR[91] R[100]mm/sec CNT100;
   1:  PR[GP1:91,1] = PR[GP1:90,1] + -23.222;
   1:  PR[GP1:91,2] = PR[GP1:90,2] + 18.152;
   1:L PR[91] R[100]mm/sec CNT100;
   1:  PR[GP1:91,1] = PR[GP1:90,1] + -23.421;
   1:  PR[GP1:91,2] = PR[GP1:90,2] + 17.997;
   1:L PR[91] R[100]mm/sec CNT100;
   1:  PR[GP1:91,1] = PR[GP1:90,1] + -27.880;
   1:  PR[GP1:91,2] = PR[GP1:90,2] + 14.749;
   1:L PR[91] R[100]mm/sec CNT100;
   1:  PR[GP1:91,1] = PR[GP1:90,1] + -28.103;
   1:  PR[GP1:91,2] = PR[GP1:90,2] + 14.508;
   1:L PR[91] R[100]mm/sec CNT100;
   1:  PR[GP1:91,1] = PR[GP1:90,1] + -31.258;
   1:  PR[GP1:91,2] = PR[GP1:90,2] + 10.591;
   1:L PR[91] R[100]mm/sec CNT100;
   1:  PR[GP1:91,1] = PR[GP1:90,1] + -31.515;
   1:  PR[GP1:91,2] = PR[GP1:90,2] + 10.200;
   1:L PR[91] R[100]mm/sec CNT100;
   1:  PR[GP1:91,1] = PR[GP1:90,1] + -33.650;
   1:  PR[GP1:91,2] = PR[GP1:90,2] + 5.344;
   1:L PR[91] R[100]mm/sec CNT100;
   1:  PR[GP1:91,1] = PR[GP1:90,1] + -33.775;
   1:  PR[GP1:91,2] = PR[GP1:90,2] + 4.861;
   1:L PR[91] R[100]mm/sec CNT100;
   1:  PR[GP1:91,1] = PR[GP1:90,1] + -33.828;
   1:  PR[GP1:91,2] = PR[GP1:90,2] + 4.192;
   1:L PR[91] R[100]mm/sec CNT100;
   1:  PR[GP1:91,1] = PR[GP1:90,1] + -34.458;
   1:  PR[GP1:91,2] = PR[GP1:90,2] + -0.354;
   1:L PR[91] R[100]mm/sec CNT100;
   1:  PR[GP1:91,1] = PR[GP1:90,1] + -34.411;
   1:  PR[GP1:91,2] = PR[GP1:90,2] + -0.953;
   1:L PR[91] R[100]mm/sec CNT100;
   1:  PR[GP1:91,1] = PR[GP1:90,1] + -33.784;
   1:  PR[GP1:91,2] = PR[GP1:90,2] + -5.449;
   1:L PR[91] R[100]mm/sec CNT100;
   1:  PR[GP1:91,1] = PR[GP1:90,1] + -33.650;
   1:  PR[GP1:91,2] = PR[GP1:90,2] + -5.968;
   1:L PR[91] R[100]mm/sec CNT100;
   1:  PR[GP1:91,1] = PR[GP1:90,1] + -33.387;
   1:  PR[GP1:91,2] = PR[GP1:90,2] + -6.552;
   1:L PR[91] R[100]mm/sec CNT100;
   1:  PR[GP1:91,1] = PR[GP1:90,1] + -31.509;
   1:  PR[GP1:91,2] = PR[GP1:90,2] + -10.835;
   1:L PR[91] R[100]mm/sec CNT100;
   1:  PR[GP1:91,1] = PR[GP1:90,1] + -31.251;
   1:  PR[GP1:91,2] = PR[GP1:90,2] + -11.226;
   1:L PR[91] R[100]mm/sec CNT100;
   1:  PR[GP1:91,1] = PR[GP1:90,1] + -28.088;
   1:  PR[GP1:91,2] = PR[GP1:90,2] + -15.146;
   1:L PR[91] R[100]mm/sec CNT100;
   1:  PR[GP1:91,1] = PR[GP1:90,1] + -27.849;
   1:  PR[GP1:91,2] = PR[GP1:90,2] + -15.405;
   1:L PR[91] R[100]mm/sec CNT100;
   1:  PR[GP1:91,1] = PR[GP1:90,1] + -27.580;
   1:  PR[GP1:91,2] = PR[GP1:90,2] + -15.615;
   1:L PR[91] R[100]mm/sec CNT100;
   1:  PR[GP1:91,1] = PR[GP1:90,1] + -23.217;
   1:  PR[GP1:91,2] = PR[GP1:90,2] + -18.778;
   1:L PR[91] R[100]mm/sec CNT100;
   1:  PR[GP1:91,1] = PR[GP1:90,1] + -23.107;
   1:  PR[GP1:91,2] = PR[GP1:90,2] + -18.840;
   1:L PR[91] R[100]mm/sec CNT100;
   1:  PR[GP1:91,1] = PR[GP1:90,1] + -17.639;
   1:  PR[GP1:91,2] = PR[GP1:90,2] + -20.967;
   1:L PR[91] R[100]mm/sec CNT100;
   1:  PR[GP1:91,1] = PR[GP1:90,1] + -15.770;
   1:  PR[GP1:91,2] = PR[GP1:90,2] + -21.191;
   1:L PR[91] R[100]mm/sec CNT100;
   1:  PR[GP1:91,1] = PR[GP1:90,1] + -11.694;
   1:  PR[GP1:91,2] = PR[GP1:90,2] + -21.719;
   1:L PR[91] R[100]mm/sec CNT100;
   1:  PR[GP1:91,1] = PR[GP1:90,1] + -11.570;
   1:  PR[GP1:91,2] = PR[GP1:90,2] + -21.707;
   1:L PR[91] R[100]mm/sec CNT100;
   1:  PR[GP1:91,1] = PR[GP1:90,1] + -5.798;
   1:  PR[GP1:91,2] = PR[GP1:90,2] + -20.969;
   1:L PR[91] R[100]mm/sec CNT100;
   1:  PR[GP1:91,1] = PR[GP1:90,1] + -5.344;
   1:  PR[GP1:91,2] = PR[GP1:90,2] + -20.811;
   1:L PR[91] R[100]mm/sec CNT100;
   1:  PR[GP1:91,1] = PR[GP1:90,1] + -1.062;
   1:  PR[GP1:91,2] = PR[GP1:90,2] + -19.120;
   1:L PR[91] R[100]mm/sec CNT100;
   1:  PR[GP1:91,1] = PR[GP1:90,1] + -0.213;
   1:  PR[GP1:91,2] = PR[GP1:90,2] + -18.976;
   1:L PR[91] R[100]mm/sec CNT100;
   1:  PR[GP1:91,1] = PR[GP1:90,1] + 0.242;
   1:  PR[GP1:91,2] = PR[GP1:90,2] + -18.818;
   1:L PR[91] R[100]mm/sec CNT100;
   1:  PR[GP1:91,1] = PR[GP1:90,1] + 1.262;
   1:  PR[GP1:91,2] = PR[GP1:90,2] + -19.131;
   1:L PR[91] R[100]mm/sec CNT100;
   1:  PR[GP1:91,1] = PR[GP1:90,1] + 2.393;
   1:  PR[GP1:91,2] = PR[GP1:90,2] + -19.593;
   1:L PR[91] R[100]mm/sec CNT100;
   1:  PR[GP1:91,1] = PR[GP1:90,1] + 5.499;
   1:  PR[GP1:91,2] = PR[GP1:90,2] + -20.809;
   1:L PR[91] R[100]mm/sec CNT100;
   1:  PR[GP1:91,1] = PR[GP1:90,1] + 5.890;
   1:  PR[GP1:91,2] = PR[GP1:90,2] + -20.947;
   1:L PR[91] R[100]mm/sec CNT100;
   1:  PR[GP1:91,1] = PR[GP1:90,1] + 11.725;
   1:  PR[GP1:91,2] = PR[GP1:90,2] + -21.707;
   1:L PR[91] R[100]mm/sec CNT100;
   1:  PR[GP1:91,1] = PR[GP1:90,1] + 11.847;
   1:  PR[GP1:91,2] = PR[GP1:90,2] + -21.719;
   1:L PR[91] R[100]mm/sec CNT100;
   1:  PR[GP1:91,1] = PR[GP1:90,1] + 15.927;
   1:  PR[GP1:91,2] = PR[GP1:90,2] + -21.190;
   1:L PR[91] R[100]mm/sec CNT100;
   1:  PR[GP1:91,1] = PR[GP1:90,1] + 17.776;
   1:  PR[GP1:91,2] = PR[GP1:90,2] + -20.975;
   1:L PR[91] R[100]mm/sec CNT100;
   1:  PR[GP1:91,1] = PR[GP1:90,1] + 23.263;
   1:  PR[GP1:91,2] = PR[GP1:90,2] + -18.842;
   1:L PR[91] R[100]mm/sec CNT100;
   1:  PR[GP1:91,1] = PR[GP1:90,1] + 23.369;
   1:  PR[GP1:91,2] = PR[GP1:90,2] + -18.782;
   1:L PR[91] R[100]mm/sec CNT100;
   1:  PR[GP1:91,1] = PR[GP1:90,1] + 28.015;
   1:  PR[GP1:91,2] = PR[GP1:90,2] + -15.395;
   1:L PR[91] R[100]mm/sec CNT100;
   1:  PR[GP1:91,1] = PR[GP1:90,1] + 28.238;
   1:  PR[GP1:91,2] = PR[GP1:90,2] + -15.155;
   1:L PR[91] R[100]mm/sec CNT100;
   1:  PR[GP1:91,1] = PR[GP1:90,1] + 31.401;
   1:  PR[GP1:91,2] = PR[GP1:90,2] + -11.227;
   1:L PR[91] R[100]mm/sec CNT100;
   1:  PR[GP1:91,1] = PR[GP1:90,1] + 31.664;
   1:  PR[GP1:91,2] = PR[GP1:90,2] + -10.830;
   1:L PR[91] R[100]mm/sec CNT100;
   1:  PR[GP1:91,1] = PR[GP1:90,1] + 33.802;
   1:  PR[GP1:91,2] = PR[GP1:90,2] + -5.997;
   1:L PR[91] R[100]mm/sec CNT100;
   1:  PR[GP1:91,1] = PR[GP1:90,1] + 33.927;
   1:  PR[GP1:91,2] = PR[GP1:90,2] + -5.522;
   1:L PR[91] R[100]mm/sec CNT100;
   1:  PR[GP1:91,1] = PR[GP1:90,1] + 33.983;
   1:  PR[GP1:91,2] = PR[GP1:90,2] + -4.834;
   1:L PR[91] R[100]mm/sec CNT100;
   1:  PR[GP1:91,1] = PR[GP1:90,1] + 34.615;
   1:  PR[GP1:91,2] = PR[GP1:90,2] + -0.271;
   1:L PR[91] R[100]mm/sec CNT100;
   1:  PR[GP1:91,1] = PR[GP1:90,1] + 34.564;
   1:  PR[GP1:91,2] = PR[GP1:90,2] + 0.352;
   1:L PR[91] R[100]mm/sec CNT100;
   1:  PR[GP1:91,1] = PR[GP1:90,1] + 33.939;
   1:  PR[GP1:91,2] = PR[GP1:90,2] + 4.854;
   1:L PR[91] R[100]mm/sec CNT100;
   1:  PR[GP1:91,1] = PR[GP1:90,1] + 33.804;
   1:  PR[GP1:91,2] = PR[GP1:90,2] + 5.368;
   1:L PR[91] R[100]mm/sec CNT100;
   1:  PR[GP1:91,1] = PR[GP1:90,1] + 31.670;
   1:  PR[GP1:91,2] = PR[GP1:90,2] + 10.195;
   1:L PR[91] R[100]mm/sec CNT100;
   1:  PR[GP1:91,1] = PR[GP1:90,1] + 31.407;
   1:  PR[GP1:91,2] = PR[GP1:90,2] + 10.593;
   1:L PR[91] R[100]mm/sec CNT100;
   1:  PR[GP1:91,1] = PR[GP1:90,1] + 28.252;
   1:  PR[GP1:91,2] = PR[GP1:90,2] + 14.517;
   1:L PR[91] R[100]mm/sec CNT100;
   1:  PR[GP1:91,1] = PR[GP1:90,1] + 28.013;
   1:  PR[GP1:91,2] = PR[GP1:90,2] + 14.775;
   1:L PR[91] R[100]mm/sec CNT100;
   1:  PR[GP1:91,1] = PR[GP1:90,1] + 27.747;
   1:  PR[GP1:91,2] = PR[GP1:90,2] + 14.982;
   1:L PR[91] R[100]mm/sec CNT100;
   1:  PR[GP1:91,1] = PR[GP1:90,1] + 23.396;
   1:  PR[GP1:91,2] = PR[GP1:90,2] + 18.144;
   1:L PR[91] R[100]mm/sec CNT100;
   1:  PR[GP1:91,1] = PR[GP1:90,1] + 23.287;
   1:  PR[GP1:91,2] = PR[GP1:90,2] + 18.205;
   1:L PR[91] R[100]mm/sec CNT100;
   1:  PR[GP1:91,1] = PR[GP1:90,1] + 17.829;
   1:  PR[GP1:91,2] = PR[GP1:90,2] + 20.334;
   1:L PR[91] R[100]mm/sec CNT100;
   1:  PR[GP1:91,1] = PR[GP1:90,1] + 15.922;
   1:  PR[GP1:91,2] = PR[GP1:90,2] + 20.566;
   1:L PR[91] R[100]mm/sec CNT100;
   1:  PR[GP1:91,1] = PR[GP1:90,1] + 11.891;
   1:  PR[GP1:91,2] = PR[GP1:90,2] + 21.095;
   1:L PR[91] R[100]mm/sec CNT100;
   1:  PR[GP1:91,1] = PR[GP1:90,1] + 11.773;
   1:  PR[GP1:91,2] = PR[GP1:90,2] + 21.084;
   1:L PR[91] R[100]mm/sec CNT100;
   1:  PR[GP1:91,1] = PR[GP1:90,1] + 6.009;
   1:  PR[GP1:91,2] = PR[GP1:90,2] + 20.357;
   1:L PR[91] R[100]mm/sec CNT100;
   1:  PR[GP1:91,1] = PR[GP1:90,1] + 5.162;
   1:  PR[GP1:91,2] = PR[GP1:90,2] + 20.054;
   1:L PR[91] R[100]mm/sec CNT100;
   1:  PR[GP1:91,1] = PR[GP1:90,1] + 1.275;
   1:  PR[GP1:91,2] = PR[GP1:90,2] + 18.503;
   1:L PR[91] R[100]mm/sec CNT100;
   1:  PR[GP1:91,1] = PR[GP1:90,1] + 0.867;
   1:  PR[GP1:91,2] = PR[GP1:90,2] + 18.398;
   1:L PR[91] R[100]mm/sec CNT100;
   1:  PR[GP1:91,1] = PR[GP1:90,1] + 0.348;
   1:  PR[GP1:91,2] = PR[GP1:90,2] + 18.189;
   1:L PR[91] R[100]mm/sec CNT100;
   1:  PR[91] = PR[90];
   1:  PR[GP1:91,1] = PR[GP1:90,1] + -1.032;
   1:  PR[GP1:91,2] = PR[GP1:90,2] + 18.674;
   1:  PR[GP1:91,3] = PR[GP1:90,3] + 43.615;
   1:L PR[91] R[100]mm/sec CNT100;
   1:  PR[GP1:91,1] = PR[GP1:90,1] + -4.434;
   1:  PR[GP1:91,2] = PR[GP1:90,2] + 20.032;
   1:L PR[91] R[100]mm/sec CNT100;
   1:  PR[GP1:91,1] = PR[GP1:90,1] + -5.639;
   1:  PR[GP1:91,2] = PR[GP1:90,2] + 20.464;
   1:L PR[91] R[100]mm/sec CNT100;
   1:  PR[GP1:91,1] = PR[GP1:90,1] + -11.157;
   1:  PR[GP1:91,2] = PR[GP1:90,2] + 21.158;
   1:L PR[91] R[100]mm/sec CNT100;
   1:  PR[GP1:91,1] = PR[GP1:90,1] + -11.538;
   1:  PR[GP1:91,2] = PR[GP1:90,2] + 21.194;
   1:L PR[91] R[100]mm/sec CNT100;
   1:  PR[GP1:91,1] = PR[GP1:90,1] + -17.433;
   1:  PR[GP1:91,2] = PR[GP1:90,2] + 20.417;
   1:L PR[91] R[100]mm/sec CNT100;
   1:  PR[GP1:91,1] = PR[GP1:90,1] + -18.873;
   1:  PR[GP1:91,2] = PR[GP1:90,2] + 19.834;
   1:L PR[91] R[100]mm/sec CNT100;
   1:  PR[GP1:91,1] = PR[GP1:90,1] + -22.962;
   1:  PR[GP1:91,2] = PR[GP1:90,2] + 18.236;
   1:L PR[91] R[100]mm/sec CNT100;
   1:  PR[GP1:91,1] = PR[GP1:90,1] + -27.684;
   1:  PR[GP1:91,2] = PR[GP1:90,2] + 14.789;
   1:L PR[91] R[100]mm/sec CNT100;
   1:  PR[GP1:91,1] = PR[GP1:90,1] + -27.807;
   1:  PR[GP1:91,2] = PR[GP1:90,2] + 14.656;
   1:L PR[91] R[100]mm/sec CNT100;
   1:  PR[GP1:91,1] = PR[GP1:90,1] + -31.122;
   1:  PR[GP1:91,2] = PR[GP1:90,2] + 10.540;
   1:L PR[91] R[100]mm/sec CNT100;
   1:  PR[GP1:91,1] = PR[GP1:90,1] + -31.300;
   1:  PR[GP1:91,2] = PR[GP1:90,2] + 10.269;
   1:L PR[91] R[100]mm/sec CNT100;
   1:  PR[GP1:91,1] = PR[GP1:90,1] + -33.475;
   1:  PR[GP1:91,2] = PR[GP1:90,2] + 5.318;
   1:L PR[91] R[100]mm/sec CNT100;
   1:  PR[GP1:91,1] = PR[GP1:90,1] + -33.565;
   1:  PR[GP1:91,2] = PR[GP1:90,2] + 4.972;
   1:L PR[91] R[100]mm/sec CNT100;
   1:  PR[GP1:91,1] = PR[GP1:90,1] + -33.607;
   1:  PR[GP1:91,2] = PR[GP1:90,2] + 4.447;
   1:L PR[91] R[100]mm/sec CNT100;
   1:  PR[GP1:91,1] = PR[GP1:90,1] + -34.272;
   1:  PR[GP1:91,2] = PR[GP1:90,2] + -0.354;
   1:L PR[91] R[100]mm/sec CNT100;
   1:  PR[GP1:91,1] = PR[GP1:90,1] + -34.236;
   1:  PR[GP1:91,2] = PR[GP1:90,2] + -0.814;
   1:L PR[91] R[100]mm/sec CNT100;
   1:  PR[GP1:91,1] = PR[GP1:90,1] + -33.574;
   1:  PR[GP1:91,2] = PR[GP1:90,2] + -5.561;
   1:L PR[91] R[100]mm/sec CNT100;
   1:  PR[GP1:91,1] = PR[GP1:90,1] + -33.475;
   1:  PR[GP1:91,2] = PR[GP1:90,2] + -5.943;
   1:L PR[91] R[100]mm/sec CNT100;
   1:  PR[GP1:91,1] = PR[GP1:90,1] + -33.272;
   1:  PR[GP1:91,2] = PR[GP1:90,2] + -6.395;
   1:L PR[91] R[100]mm/sec CNT100;
   1:  PR[GP1:91,1] = PR[GP1:90,1] + -31.293;
   1:  PR[GP1:91,2] = PR[GP1:90,2] + -10.905;
   1:L PR[91] R[100]mm/sec CNT100;
   1:  PR[GP1:91,1] = PR[GP1:90,1] + -31.115;
   1:  PR[GP1:91,2] = PR[GP1:90,2] + -11.175;
   1:L PR[91] R[100]mm/sec CNT100;
   1:  PR[GP1:91,1] = PR[GP1:90,1] + -27.792;
   1:  PR[GP1:91,2] = PR[GP1:90,2] + -15.295;
   1:L PR[91] R[100]mm/sec CNT100;
   1:  PR[GP1:91,1] = PR[GP1:90,1] + -27.652;
   1:  PR[GP1:91,2] = PR[GP1:90,2] + -15.446;
   1:L PR[91] R[100]mm/sec CNT100;
   1:  PR[GP1:91,1] = PR[GP1:90,1] + -27.491;
   1:  PR[GP1:91,2] = PR[GP1:90,2] + -15.571;
   1:L PR[91] R[100]mm/sec CNT100;
   1:  PR[GP1:91,1] = PR[GP1:90,1] + -22.937;
   1:  PR[GP1:91,2] = PR[GP1:90,2] + -18.873;
   1:L PR[91] R[100]mm/sec CNT100;
   1:  PR[GP1:91,1] = PR[GP1:90,1] + -18.876;
   1:  PR[GP1:91,2] = PR[GP1:90,2] + -20.454;
   1:L PR[91] R[100]mm/sec CNT100;
   1:  PR[GP1:91,1] = PR[GP1:90,1] + -17.397;
   1:  PR[GP1:91,2] = PR[GP1:90,2] + -21.050;
   1:L PR[91] R[100]mm/sec CNT100;
   1:  PR[GP1:91,1] = PR[GP1:90,1] + -11.494;
   1:  PR[GP1:91,2] = PR[GP1:90,2] + -21.818;
   1:L PR[91] R[100]mm/sec CNT100;
   1:  PR[GP1:91,1] = PR[GP1:90,1] + -11.105;
   1:  PR[GP1:91,2] = PR[GP1:90,2] + -21.780;
   1:L PR[91] R[100]mm/sec CNT100;
   1:  PR[GP1:91,1] = PR[GP1:90,1] + -5.581;
   1:  PR[GP1:91,2] = PR[GP1:90,2] + -21.074;
   1:L PR[91] R[100]mm/sec CNT100;
   1:  PR[GP1:91,1] = PR[GP1:90,1] + -4.908;
   1:  PR[GP1:91,2] = PR[GP1:90,2] + -20.839;
   1:L PR[91] R[100]mm/sec CNT100;
   1:  PR[GP1:91,1] = PR[GP1:90,1] + -1.041;
   1:  PR[GP1:91,2] = PR[GP1:90,2] + -19.323;
   1:L PR[91] R[100]mm/sec CNT100;
   1:  PR[GP1:91,1] = PR[GP1:90,1] + 0.382;
   1:  PR[GP1:91,2] = PR[GP1:90,2] + -19.085;
   1:L PR[91] R[100]mm/sec CNT100;
   1:  PR[GP1:91,1] = PR[GP1:90,1] + 1.281;
   1:  PR[GP1:91,2] = PR[GP1:90,2] + -19.357;
   1:L PR[91] R[100]mm/sec CNT100;
   1:  PR[GP1:91,1] = PR[GP1:90,1] + 5.065;
   1:  PR[GP1:91,2] = PR[GP1:90,2] + -20.838;
   1:L PR[91] R[100]mm/sec CNT100;
   1:  PR[GP1:91,1] = PR[GP1:90,1] + 5.652;
   1:  PR[GP1:91,2] = PR[GP1:90,2] + -21.045;
   1:L PR[91] R[100]mm/sec CNT100;
   1:  PR[GP1:91,1] = PR[GP1:90,1] + 11.261;
   1:  PR[GP1:91,2] = PR[GP1:90,2] + -21.780;
   1:L PR[91] R[100]mm/sec CNT100;
   1:  PR[GP1:91,1] = PR[GP1:90,1] + 11.648;
   1:  PR[GP1:91,2] = PR[GP1:90,2] + -21.819;
   1:L PR[91] R[100]mm/sec CNT100;
   1:  PR[GP1:91,1] = PR[GP1:90,1] + 17.552;
   1:  PR[GP1:91,2] = PR[GP1:90,2] + -21.050;
   1:L PR[91] R[100]mm/sec CNT100;
   1:  PR[GP1:91,1] = PR[GP1:90,1] + 19.031;
   1:  PR[GP1:91,2] = PR[GP1:90,2] + -20.454;
   1:L PR[91] R[100]mm/sec CNT100;
   1:  PR[GP1:91,1] = PR[GP1:90,1] + 23.091;
   1:  PR[GP1:91,2] = PR[GP1:90,2] + -18.876;
   1:L PR[91] R[100]mm/sec CNT100;
   1:  PR[GP1:91,1] = PR[GP1:90,1] + 27.820;
   1:  PR[GP1:91,2] = PR[GP1:90,2] + -15.434;
   1:L PR[91] R[100]mm/sec CNT100;
   1:  PR[GP1:91,1] = PR[GP1:90,1] + 27.943;
   1:  PR[GP1:91,2] = PR[GP1:90,2] + -15.301;
   1:L PR[91] R[100]mm/sec CNT100;
   1:  PR[GP1:91,1] = PR[GP1:90,1] + 31.267;
   1:  PR[GP1:91,2] = PR[GP1:90,2] + -11.174;
   1:L PR[91] R[100]mm/sec CNT100;
   1:  PR[GP1:91,1] = PR[GP1:90,1] + 31.449;
   1:  PR[GP1:91,2] = PR[GP1:90,2] + -10.899;
   1:L PR[91] R[100]mm/sec CNT100;
   1:  PR[GP1:91,1] = PR[GP1:90,1] + 33.628;
   1:  PR[GP1:91,2] = PR[GP1:90,2] + -5.970;
   1:L PR[91] R[100]mm/sec CNT100;
   1:  PR[GP1:91,1] = PR[GP1:90,1] + 33.717;
   1:  PR[GP1:91,2] = PR[GP1:90,2] + -5.630;
   1:L PR[91] R[100]mm/sec CNT100;
   1:  PR[GP1:91,1] = PR[GP1:90,1] + 33.762;
   1:  PR[GP1:91,2] = PR[GP1:90,2] + -5.090;
   1:L PR[91] R[100]mm/sec CNT100;
   1:  PR[GP1:91,1] = PR[GP1:90,1] + 34.429;
   1:  PR[GP1:91,2] = PR[GP1:90,2] + -0.271;
   1:L PR[91] R[100]mm/sec CNT100;
   1:  PR[GP1:91,1] = PR[GP1:90,1] + 34.390;
   1:  PR[GP1:91,2] = PR[GP1:90,2] + 0.208;
   1:L PR[91] R[100]mm/sec CNT100;
   1:  PR[GP1:91,1] = PR[GP1:90,1] + 33.729;
   1:  PR[GP1:91,2] = PR[GP1:90,2] + 4.961;
   1:L PR[91] R[100]mm/sec CNT100;
   1:  PR[GP1:91,1] = PR[GP1:90,1] + 33.630;
   1:  PR[GP1:91,2] = PR[GP1:90,2] + 5.340;
   1:L PR[91] R[100]mm/sec CNT100;
   1:  PR[GP1:91,1] = PR[GP1:90,1] + 31.456;
   1:  PR[GP1:91,2] = PR[GP1:90,2] + 10.264;
   1:L PR[91] R[100]mm/sec CNT100;
   1:  PR[GP1:91,1] = PR[GP1:90,1] + 31.273;
   1:  PR[GP1:91,2] = PR[GP1:90,2] + 10.539;
   1:L PR[91] R[100]mm/sec CNT100;
   1:  PR[GP1:91,1] = PR[GP1:90,1] + 27.958;
   1:  PR[GP1:91,2] = PR[GP1:90,2] + 14.663;
   1:L PR[91] R[100]mm/sec CNT100;
   1:  PR[GP1:91,1] = PR[GP1:90,1] + 27.819;
   1:  PR[GP1:91,2] = PR[GP1:90,2] + 14.813;
   1:L PR[91] R[100]mm/sec CNT100;
   1:  PR[GP1:91,1] = PR[GP1:90,1] + 27.660;
   1:  PR[GP1:91,2] = PR[GP1:90,2] + 14.937;
   1:L PR[91] R[100]mm/sec CNT100;
   1:  PR[GP1:91,1] = PR[GP1:90,1] + 23.117;
   1:  PR[GP1:91,2] = PR[GP1:90,2] + 18.238;
   1:L PR[91] R[100]mm/sec CNT100;
   1:  PR[GP1:91,1] = PR[GP1:90,1] + 19.030;
   1:  PR[GP1:91,2] = PR[GP1:90,2] + 19.834;
   1:L PR[91] R[100]mm/sec CNT100;
   1:  PR[GP1:91,1] = PR[GP1:90,1] + 17.587;
   1:  PR[GP1:91,2] = PR[GP1:90,2] + 20.417;
   1:L PR[91] R[100]mm/sec CNT100;
   1:  PR[GP1:91,1] = PR[GP1:90,1] + 11.691;
   1:  PR[GP1:91,2] = PR[GP1:90,2] + 21.195;
   1:L PR[91] R[100]mm/sec CNT100;
   1:  PR[GP1:91,1] = PR[GP1:90,1] + 11.311;
   1:  PR[GP1:91,2] = PR[GP1:90,2] + 21.158;
   1:L PR[91] R[100]mm/sec CNT100;
   1:  PR[GP1:91,1] = PR[GP1:90,1] + 5.793;
   1:  PR[GP1:91,2] = PR[GP1:90,2] + 20.462;
   1:L PR[91] R[100]mm/sec CNT100;
   1:  PR[GP1:91,1] = PR[GP1:90,1] + 4.587;
   1:  PR[GP1:91,2] = PR[GP1:90,2] + 20.030;
   1:L PR[91] R[100]mm/sec CNT100;
   1:  PR[GP1:91,1] = PR[GP1:90,1] + 1.261;
   1:  PR[GP1:91,2] = PR[GP1:90,2] + 18.703;
   1:L PR[91] R[100]mm/sec CNT100;
   1:  PR[GP1:91,1] = PR[GP1:90,1] + 0.369;
   1:  PR[GP1:91,2] = PR[GP1:90,2] + 18.470;
   1:L PR[91] R[100]mm/sec CNT100;
   1:  PR[91] = PR[90];
   1:  PR[GP1:91,1] = PR[GP1:90,1] + -1.017;
   1:  PR[GP1:91,2] = PR[GP1:90,2] + 18.874;
   1:  PR[GP1:91,3] = PR[GP1:90,3] + 44.225;
   1:L PR[91] R[100]mm/sec CNT100;
   1:  PR[GP1:91,1] = PR[GP1:90,1] + -3.858;
   1:  PR[GP1:91,2] = PR[GP1:90,2] + 20.009;
   1:L PR[91] R[100]mm/sec CNT100;
   1:  PR[GP1:91,1] = PR[GP1:90,1] + -5.422;
   1:  PR[GP1:91,2] = PR[GP1:90,2] + 20.569;
   1:L PR[91] R[100]mm/sec CNT100;
   1:  PR[GP1:91,1] = PR[GP1:90,1] + -10.694;
   1:  PR[GP1:91,2] = PR[GP1:90,2] + 21.232;
   1:L PR[91] R[100]mm/sec CNT100;
   1:  PR[GP1:91,1] = PR[GP1:90,1] + -11.339;
   1:  PR[GP1:91,2] = PR[GP1:90,2] + 21.294;
   1:L PR[91] R[100]mm/sec CNT100;
   1:  PR[GP1:91,1] = PR[GP1:90,1] + -17.031;
   1:  PR[GP1:91,2] = PR[GP1:90,2] + 20.547;
   1:L PR[91] R[100]mm/sec CNT100;
   1:  PR[GP1:91,1] = PR[GP1:90,1] + -17.231;
   1:  PR[GP1:91,2] = PR[GP1:90,2] + 20.514;
   1:L PR[91] R[100]mm/sec CNT100;
   1:  PR[GP1:91,1] = PR[GP1:90,1] + -22.722;
   1:  PR[GP1:91,2] = PR[GP1:90,2] + 18.298;
   1:L PR[91] R[100]mm/sec CNT100;
   1:  PR[GP1:91,1] = PR[GP1:90,1] + -27.488;
   1:  PR[GP1:91,2] = PR[GP1:90,2] + 14.829;
   1:L PR[91] R[100]mm/sec CNT100;
   1:  PR[GP1:91,1] = PR[GP1:90,1] + -27.511;
   1:  PR[GP1:91,2] = PR[GP1:90,2] + 14.804;
   1:L PR[91] R[100]mm/sec CNT100;
   1:  PR[GP1:91,1] = PR[GP1:90,1] + -30.986;
   1:  PR[GP1:91,2] = PR[GP1:90,2] + 10.489;
   1:L PR[91] R[100]mm/sec CNT100;
   1:  PR[GP1:91,1] = PR[GP1:90,1] + -31.085;
   1:  PR[GP1:91,2] = PR[GP1:90,2] + 10.338;
   1:L PR[91] R[100]mm/sec CNT100;
   1:  PR[GP1:91,1] = PR[GP1:90,1] + -33.300;
   1:  PR[GP1:91,2] = PR[GP1:90,2] + 5.293;
   1:L PR[91] R[100]mm/sec CNT100;
   1:  PR[GP1:91,1] = PR[GP1:90,1] + -33.354;
   1:  PR[GP1:91,2] = PR[GP1:90,2] + 5.083;
   1:L PR[91] R[100]mm/sec CNT100;
   1:  PR[GP1:91,1] = PR[GP1:90,1] + -33.385;
   1:  PR[GP1:91,2] = PR[GP1:90,2] + 4.702;
   1:L PR[91] R[100]mm/sec CNT100;
   1:  PR[GP1:91,1] = PR[GP1:90,1] + -34.086;
   1:  PR[GP1:91,2] = PR[GP1:90,2] + -0.354;
   1:L PR[91] R[100]mm/sec CNT100;
   1:  PR[GP1:91,1] = PR[GP1:90,1] + -34.060;
   1:  PR[GP1:91,2] = PR[GP1:90,2] + -0.674;
   1:L PR[91] R[100]mm/sec CNT100;
   1:  PR[GP1:91,1] = PR[GP1:90,1] + -33.363;
   1:  PR[GP1:91,2] = PR[GP1:90,2] + -5.673;
   1:L PR[91] R[100]mm/sec CNT100;
   1:  PR[GP1:91,1] = PR[GP1:90,1] + -33.300;
   1:  PR[GP1:91,2] = PR[GP1:90,2] + -5.917;
   1:L PR[91] R[100]mm/sec CNT100;
   1:  PR[GP1:91,1] = PR[GP1:90,1] + -33.156;
   1:  PR[GP1:91,2] = PR[GP1:90,2] + -6.238;
   1:L PR[91] R[100]mm/sec CNT100;
   1:  PR[GP1:91,1] = PR[GP1:90,1] + -31.078;
   1:  PR[GP1:91,2] = PR[GP1:90,2] + -10.975;
   1:L PR[91] R[100]mm/sec CNT100;
   1:  PR[GP1:91,1] = PR[GP1:90,1] + -30.980;
   1:  PR[GP1:91,2] = PR[GP1:90,2] + -11.125;
   1:L PR[91] R[100]mm/sec CNT100;
   1:  PR[GP1:91,1] = PR[GP1:90,1] + -27.495;
   1:  PR[GP1:91,2] = PR[GP1:90,2] + -15.443;
   1:L PR[91] R[100]mm/sec CNT100;
   1:  PR[GP1:91,1] = PR[GP1:90,1] + -27.473;
   1:  PR[GP1:91,2] = PR[GP1:90,2] + -15.467;
   1:L PR[91] R[100]mm/sec CNT100;
   1:  PR[GP1:91,1] = PR[GP1:90,1] + -22.696;
   1:  PR[GP1:91,2] = PR[GP1:90,2] + -18.937;
   1:L PR[91] R[100]mm/sec CNT100;
   1:  PR[GP1:91,1] = PR[GP1:90,1] + -17.195;
   1:  PR[GP1:91,2] = PR[GP1:90,2] + -21.148;
   1:L PR[91] R[100]mm/sec CNT100;
   1:  PR[GP1:91,1] = PR[GP1:90,1] + -16.992;
   1:  PR[GP1:91,2] = PR[GP1:90,2] + -21.180;
   1:L PR[91] R[100]mm/sec CNT100;
   1:  PR[GP1:91,1] = PR[GP1:90,1] + -11.296;
   1:  PR[GP1:91,2] = PR[GP1:90,2] + -21.918;
   1:L PR[91] R[100]mm/sec CNT100;
   1:  PR[GP1:91,1] = PR[GP1:90,1] + -10.640;
   1:  PR[GP1:91,2] = PR[GP1:90,2] + -21.853;
   1:L PR[91] R[100]mm/sec CNT100;
   1:  PR[GP1:91,1] = PR[GP1:90,1] + -5.365;
   1:  PR[GP1:91,2] = PR[GP1:90,2] + -21.179;
   1:L PR[91] R[100]mm/sec CNT100;
   1:  PR[GP1:91,1] = PR[GP1:90,1] + -4.473;
   1:  PR[GP1:91,2] = PR[GP1:90,2] + -20.868;
   1:L PR[91] R[100]mm/sec CNT100;
   1:  PR[GP1:91,1] = PR[GP1:90,1] + -1.022;
   1:  PR[GP1:91,2] = PR[GP1:90,2] + -19.515;
   1:L PR[91] R[100]mm/sec CNT100;
   1:  PR[GP1:91,1] = PR[GP1:90,1] + 0.411;
   1:  PR[GP1:91,2] = PR[GP1:90,2] + -19.282;
   1:L PR[91] R[100]mm/sec CNT100;
   1:  PR[GP1:91,1] = PR[GP1:90,1] + 1.272;
   1:  PR[GP1:91,2] = PR[GP1:90,2] + -19.552;
   1:L PR[91] R[100]mm/sec CNT100;
   1:  PR[GP1:91,1] = PR[GP1:90,1] + 4.630;
   1:  PR[GP1:91,2] = PR[GP1:90,2] + -20.867;
   1:L PR[91] R[100]mm/sec CNT100;
   1:  PR[GP1:91,1] = PR[GP1:90,1] + 5.411;
   1:  PR[GP1:91,2] = PR[GP1:90,2] + -21.143;
   1:L PR[91] R[100]mm/sec CNT100;
   1:  PR[GP1:91,1] = PR[GP1:90,1] + 10.700;
   1:  PR[GP1:91,2] = PR[GP1:90,2] + -21.827;
   1:L PR[91] R[100]mm/sec CNT100;
   1:  PR[GP1:91,1] = PR[GP1:90,1] + 10.853;
   1:  PR[GP1:91,2] = PR[GP1:90,2] + -21.859;
   1:L PR[91] R[100]mm/sec CNT100;
   1:  PR[GP1:91,1] = PR[GP1:90,1] + 11.450;
   1:  PR[GP1:91,2] = PR[GP1:90,2] + -21.918;
   1:L PR[91] R[100]mm/sec CNT100;
   1:  PR[GP1:91,1] = PR[GP1:90,1] + 17.146;
   1:  PR[GP1:91,2] = PR[GP1:90,2] + -21.180;
   1:L PR[91] R[100]mm/sec CNT100;
   1:  PR[GP1:91,1] = PR[GP1:90,1] + 17.349;
   1:  PR[GP1:91,2] = PR[GP1:90,2] + -21.148;
   1:L PR[91] R[100]mm/sec CNT100;
   1:  PR[GP1:91,1] = PR[GP1:90,1] + 22.851;
   1:  PR[GP1:91,2] = PR[GP1:90,2] + -18.939;
   1:L PR[91] R[100]mm/sec CNT100;
   1:  PR[GP1:91,1] = PR[GP1:90,1] + 27.626;
   1:  PR[GP1:91,2] = PR[GP1:90,2] + -15.472;
   1:L PR[91] R[100]mm/sec CNT100;
   1:  PR[GP1:91,1] = PR[GP1:90,1] + 27.648;
   1:  PR[GP1:91,2] = PR[GP1:90,2] + -15.448;
   1:L PR[91] R[100]mm/sec CNT100;
   1:  PR[GP1:91,1] = PR[GP1:90,1] + 31.132;
   1:  PR[GP1:91,2] = PR[GP1:90,2] + -11.122;
   1:L PR[91] R[100]mm/sec CNT100;
   1:  PR[GP1:91,1] = PR[GP1:90,1] + 31.234;
   1:  PR[GP1:91,2] = PR[GP1:90,2] + -10.967;
   1:L PR[91] R[100]mm/sec CNT100;
   1:  PR[GP1:91,1] = PR[GP1:90,1] + 33.454;
   1:  PR[GP1:91,2] = PR[GP1:90,2] + -5.943;
   1:L PR[91] R[100]mm/sec CNT100;
   1:  PR[GP1:91,1] = PR[GP1:90,1] + 33.508;
   1:  PR[GP1:91,2] = PR[GP1:90,2] + -5.738;
   1:L PR[91] R[100]mm/sec CNT100;
   1:  PR[GP1:91,1] = PR[GP1:90,1] + 33.540;
   1:  PR[GP1:91,2] = PR[GP1:90,2] + -5.345;
   1:L PR[91] R[100]mm/sec CNT100;
   1:  PR[GP1:91,1] = PR[GP1:90,1] + 34.242;
   1:  PR[GP1:91,2] = PR[GP1:90,2] + -0.271;
   1:L PR[91] R[100]mm/sec CNT100;
   1:  PR[GP1:91,1] = PR[GP1:90,1] + 34.215;
   1:  PR[GP1:91,2] = PR[GP1:90,2] + 0.065;
   1:L PR[91] R[100]mm/sec CNT100;
   1:  PR[GP1:91,1] = PR[GP1:90,1] + 33.520;
   1:  PR[GP1:91,2] = PR[GP1:90,2] + 5.069;
   1:L PR[91] R[100]mm/sec CNT100;
   1:  PR[GP1:91,1] = PR[GP1:90,1] + 33.456;
   1:  PR[GP1:91,2] = PR[GP1:90,2] + 5.313;
   1:L PR[91] R[100]mm/sec CNT100;
   1:  PR[GP1:91,1] = PR[GP1:90,1] + 31.241;
   1:  PR[GP1:91,2] = PR[GP1:90,2] + 10.332;
   1:L PR[91] R[100]mm/sec CNT100;
   1:  PR[GP1:91,1] = PR[GP1:90,1] + 31.139;
   1:  PR[GP1:91,2] = PR[GP1:90,2] + 10.487;
   1:L PR[91] R[100]mm/sec CNT100;
   1:  PR[GP1:91,1] = PR[GP1:90,1] + 27.664;
   1:  PR[GP1:91,2] = PR[GP1:90,2] + 14.809;
   1:L PR[91] R[100]mm/sec CNT100;
   1:  PR[GP1:91,1] = PR[GP1:90,1] + 27.641;
   1:  PR[GP1:91,2] = PR[GP1:90,2] + 14.834;
   1:L PR[91] R[100]mm/sec CNT100;
   1:  PR[GP1:91,1] = PR[GP1:90,1] + 22.877;
   1:  PR[GP1:91,2] = PR[GP1:90,2] + 18.301;
   1:L PR[91] R[100]mm/sec CNT100;
   1:  PR[GP1:91,1] = PR[GP1:90,1] + 17.385;
   1:  PR[GP1:91,2] = PR[GP1:90,2] + 20.514;
   1:L PR[91] R[100]mm/sec CNT100;
   1:  PR[GP1:91,1] = PR[GP1:90,1] + 17.184;
   1:  PR[GP1:91,2] = PR[GP1:90,2] + 20.547;
   1:L PR[91] R[100]mm/sec CNT100;
   1:  PR[GP1:91,1] = PR[GP1:90,1] + 11.493;
   1:  PR[GP1:91,2] = PR[GP1:90,2] + 21.294;
   1:L PR[91] R[100]mm/sec CNT100;
   1:  PR[GP1:91,1] = PR[GP1:90,1] + 10.848;
   1:  PR[GP1:91,2] = PR[GP1:90,2] + 21.232;
   1:L PR[91] R[100]mm/sec CNT100;
   1:  PR[GP1:91,1] = PR[GP1:90,1] + 5.555;
   1:  PR[GP1:91,2] = PR[GP1:90,2] + 20.565;
   1:L PR[91] R[100]mm/sec CNT100;
   1:  PR[GP1:91,1] = PR[GP1:90,1] + 5.340;
   1:  PR[GP1:91,2] = PR[GP1:90,2] + 20.494;
   1:L PR[91] R[100]mm/sec CNT100;
   1:  PR[GP1:91,1] = PR[GP1:90,1] + 4.017;
   1:  PR[GP1:91,2] = PR[GP1:90,2] + 20.009;
   1:L PR[91] R[100]mm/sec CNT100;
   1:  PR[GP1:91,1] = PR[GP1:90,1] + 1.242;
   1:  PR[GP1:91,2] = PR[GP1:90,2] + 18.902;
   1:L PR[91] R[100]mm/sec CNT100;
   1:  PR[GP1:91,1] = PR[GP1:90,1] + 0.855;
   1:  PR[GP1:91,2] = PR[GP1:90,2] + 18.802;
   1:L PR[91] R[100]mm/sec CNT100;
   1:  PR[GP1:91,1] = PR[GP1:90,1] + 0.519;
   1:  PR[GP1:91,2] = PR[GP1:90,2] + 18.647;
   1:L PR[91] R[100]mm/sec CNT100;
   1:  PR[91] = PR[90];
   1:  PR[GP1:91,1] = PR[GP1:90,1] + -1.002;
   1:  PR[GP1:91,2] = PR[GP1:90,2] + 19.074;
   1:  PR[GP1:91,3] = PR[GP1:90,3] + 44.835;
   1:L PR[91] R[100]mm/sec CNT100;
   1:  PR[GP1:91,1] = PR[GP1:90,1] + -3.287;
   1:  PR[GP1:91,2] = PR[GP1:90,2] + 19.987;
   1:L PR[91] R[100]mm/sec CNT100;
   1:  PR[GP1:91,1] = PR[GP1:90,1] + -5.044;
   1:  PR[GP1:91,2] = PR[GP1:90,2] + 20.628;
   1:L PR[91] R[100]mm/sec CNT100;
   1:  PR[GP1:91,1] = PR[GP1:90,1] + -5.181;
   1:  PR[GP1:91,2] = PR[GP1:90,2] + 20.671;
   1:L PR[91] R[100]mm/sec CNT100;
   1:  PR[GP1:91,1] = PR[GP1:90,1] + -10.231;
   1:  PR[GP1:91,2] = PR[GP1:90,2] + 21.306;
   1:L PR[91] R[100]mm/sec CNT100;
   1:  PR[GP1:91,1] = PR[GP1:90,1] + -11.140;
   1:  PR[GP1:91,2] = PR[GP1:90,2] + 21.393;
   1:L PR[91] R[100]mm/sec CNT100;
   1:  PR[GP1:91,1] = PR[GP1:90,1] + -16.581;
   1:  PR[GP1:91,2] = PR[GP1:90,2] + 20.679;
   1:L PR[91] R[100]mm/sec CNT100;
   1:  PR[GP1:91,1] = PR[GP1:90,1] + -17.045;
   1:  PR[GP1:91,2] = PR[GP1:90,2] + 20.605;
   1:L PR[91] R[100]mm/sec CNT100;
   1:  PR[GP1:91,1] = PR[GP1:90,1] + -22.543;
   1:  PR[GP1:91,2] = PR[GP1:90,2] + 18.372;
   1:L PR[91] R[100]mm/sec CNT100;
   1:  PR[GP1:91,1] = PR[GP1:90,1] + -25.480;
   1:  PR[GP1:91,2] = PR[GP1:90,2] + 16.189;
   1:L PR[91] R[100]mm/sec CNT100;
   1:  PR[GP1:91,1] = PR[GP1:90,1] + -27.252;
   1:  PR[GP1:91,2] = PR[GP1:90,2] + 14.898;
   1:L PR[91] R[100]mm/sec CNT100;
   1:  PR[GP1:91,1] = PR[GP1:90,1] + -30.851;
   1:  PR[GP1:91,2] = PR[GP1:90,2] + 10.438;
   1:L PR[91] R[100]mm/sec CNT100;
   1:  PR[GP1:91,1] = PR[GP1:90,1] + -30.874;
   1:  PR[GP1:91,2] = PR[GP1:90,2] + 10.403;
   1:L PR[91] R[100]mm/sec CNT100;
   1:  PR[GP1:91,1] = PR[GP1:90,1] + -30.924;
   1:  PR[GP1:91,2] = PR[GP1:90,2] + 10.292;
   1:L PR[91] R[100]mm/sec CNT100;
   1:  PR[GP1:91,1] = PR[GP1:90,1] + -33.125;
   1:  PR[GP1:91,2] = PR[GP1:90,2] + 5.268;
   1:L PR[91] R[100]mm/sec CNT100;
   1:  PR[GP1:91,1] = PR[GP1:90,1] + -33.144;
   1:  PR[GP1:91,2] = PR[GP1:90,2] + 5.195;
   1:L PR[91] R[100]mm/sec CNT100;
   1:  PR[GP1:91,1] = PR[GP1:90,1] + -33.163;
   1:  PR[GP1:91,2] = PR[GP1:90,2] + 4.957;
   1:L PR[91] R[100]mm/sec CNT100;
   1:  PR[GP1:91,1] = PR[GP1:90,1] + -33.900;
   1:  PR[GP1:91,2] = PR[GP1:90,2] + -0.354;
   1:L PR[91] R[100]mm/sec CNT100;
   1:  PR[GP1:91,1] = PR[GP1:90,1] + -33.885;
   1:  PR[GP1:91,2] = PR[GP1:90,2] + -0.535;
   1:L PR[91] R[100]mm/sec CNT100;
   1:  PR[GP1:91,1] = PR[GP1:90,1] + -33.153;
   1:  PR[GP1:91,2] = PR[GP1:90,2] + -5.784;
   1:L PR[91] R[100]mm/sec CNT100;
   1:  PR[GP1:91,1] = PR[GP1:90,1] + -33.125;
   1:  PR[GP1:91,2] = PR[GP1:90,2] + -5.892;
   1:L PR[91] R[100]mm/sec CNT100;
   1:  PR[GP1:91,1] = PR[GP1:90,1] + -33.040;
   1:  PR[GP1:91,2] = PR[GP1:90,2] + -6.081;
   1:L PR[91] R[100]mm/sec CNT100;
   1:  PR[GP1:91,1] = PR[GP1:90,1] + -30.863;
   1:  PR[GP1:91,2] = PR[GP1:90,2] + -11.044;
   1:L PR[91] R[100]mm/sec CNT100;
   1:  PR[GP1:91,1] = PR[GP1:90,1] + -30.844;
   1:  PR[GP1:91,2] = PR[GP1:90,2] + -11.074;
   1:L PR[91] R[100]mm/sec CNT100;
   1:  PR[GP1:91,1] = PR[GP1:90,1] + -27.236;
   1:  PR[GP1:91,2] = PR[GP1:90,2] + -15.537;
   1:L PR[91] R[100]mm/sec CNT100;
   1:  PR[GP1:91,1] = PR[GP1:90,1] + -25.483;
   1:  PR[GP1:91,2] = PR[GP1:90,2] + -16.812;
   1:L PR[91] R[100]mm/sec CNT100;
   1:  PR[GP1:91,1] = PR[GP1:90,1] + -22.517;
   1:  PR[GP1:91,2] = PR[GP1:90,2] + -19.010;
   1:L PR[91] R[100]mm/sec CNT100;
   1:  PR[GP1:91,1] = PR[GP1:90,1] + -17.009;
   1:  PR[GP1:91,2] = PR[GP1:90,2] + -21.238;
   1:L PR[91] R[100]mm/sec CNT100;
   1:  PR[GP1:91,1] = PR[GP1:90,1] + -16.542;
   1:  PR[GP1:91,2] = PR[GP1:90,2] + -21.312;
   1:L PR[91] R[100]mm/sec CNT100;
   1:  PR[GP1:91,1] = PR[GP1:90,1] + -11.097;
   1:  PR[GP1:91,2] = PR[GP1:90,2] + -22.018;
   1:L PR[91] R[100]mm/sec CNT100;
   1:  PR[GP1:91,1] = PR[GP1:90,1] + -10.175;
   1:  PR[GP1:91,2] = PR[GP1:90,2] + -21.926;
   1:L PR[91] R[100]mm/sec CNT100;
   1:  PR[GP1:91,1] = PR[GP1:90,1] + -5.149;
   1:  PR[GP1:91,2] = PR[GP1:90,2] + -21.284;
   1:L PR[91] R[100]mm/sec CNT100;
   1:  PR[GP1:91,1] = PR[GP1:90,1] + -4.038;
   1:  PR[GP1:91,2] = PR[GP1:90,2] + -20.897;
   1:L PR[91] R[100]mm/sec CNT100;
   1:  PR[GP1:91,1] = PR[GP1:90,1] + -1.002;
   1:  PR[GP1:91,2] = PR[GP1:90,2] + -19.707;
   1:L PR[91] R[100]mm/sec CNT100;
   1:  PR[GP1:91,1] = PR[GP1:90,1] + 0.577;
   1:  PR[GP1:91,2] = PR[GP1:90,2] + -19.458;
   1:L PR[91] R[100]mm/sec CNT100;
   1:  PR[GP1:91,1] = PR[GP1:90,1] + 0.929;
   1:  PR[GP1:91,2] = PR[GP1:90,2] + -19.646;
   1:L PR[91] R[100]mm/sec CNT100;
   1:  PR[GP1:91,1] = PR[GP1:90,1] + 1.247;
   1:  PR[GP1:91,2] = PR[GP1:90,2] + -19.742;
   1:L PR[91] R[100]mm/sec CNT100;
   1:  PR[GP1:91,1] = PR[GP1:90,1] + 4.196;
   1:  PR[GP1:91,2] = PR[GP1:90,2] + -20.896;
   1:L PR[91] R[100]mm/sec CNT100;
   1:  PR[GP1:91,1] = PR[GP1:90,1] + 5.172;
   1:  PR[GP1:91,2] = PR[GP1:90,2] + -21.240;
   1:L PR[91] R[100]mm/sec CNT100;
   1:  PR[GP1:91,1] = PR[GP1:90,1] + 10.180;
   1:  PR[GP1:91,2] = PR[GP1:90,2] + -21.888;
   1:L PR[91] R[100]mm/sec CNT100;
   1:  PR[GP1:91,1] = PR[GP1:90,1] + 10.388;
   1:  PR[GP1:91,2] = PR[GP1:90,2] + -21.932;
   1:L PR[91] R[100]mm/sec CNT100;
   1:  PR[GP1:91,1] = PR[GP1:90,1] + 11.251;
   1:  PR[GP1:91,2] = PR[GP1:90,2] + -22.018;
   1:L PR[91] R[100]mm/sec CNT100;
   1:  PR[GP1:91,1] = PR[GP1:90,1] + 16.697;
   1:  PR[GP1:91,2] = PR[GP1:90,2] + -21.312;
   1:L PR[91] R[100]mm/sec CNT100;
   1:  PR[GP1:91,1] = PR[GP1:90,1] + 17.164;
   1:  PR[GP1:91,2] = PR[GP1:90,2] + -21.238;
   1:L PR[91] R[100]mm/sec CNT100;
   1:  PR[GP1:91,1] = PR[GP1:90,1] + 22.673;
   1:  PR[GP1:91,2] = PR[GP1:90,2] + -19.012;
   1:L PR[91] R[100]mm/sec CNT100;
   1:  PR[GP1:91,1] = PR[GP1:90,1] + 25.638;
   1:  PR[GP1:91,2] = PR[GP1:90,2] + -16.814;
   1:L PR[91] R[100]mm/sec CNT100;
   1:  PR[GP1:91,1] = PR[GP1:90,1] + 27.390;
   1:  PR[GP1:91,2] = PR[GP1:90,2] + -15.541;
   1:L PR[91] R[100]mm/sec CNT100;
   1:  PR[GP1:91,1] = PR[GP1:90,1] + 30.998;
   1:  PR[GP1:91,2] = PR[GP1:90,2] + -11.069;
   1:L PR[91] R[100]mm/sec CNT100;
   1:  PR[GP1:91,1] = PR[GP1:90,1] + 31.020;
   1:  PR[GP1:91,2] = PR[GP1:90,2] + -11.036;
   1:L PR[91] R[100]mm/sec CNT100;
   1:  PR[GP1:91,1] = PR[GP1:90,1] + 33.280;
   1:  PR[GP1:91,2] = PR[GP1:90,2] + -5.916;
   1:L PR[91] R[100]mm/sec CNT100;
   1:  PR[GP1:91,1] = PR[GP1:90,1] + 33.298;
   1:  PR[GP1:91,2] = PR[GP1:90,2] + -5.846;
   1:L PR[91] R[100]mm/sec CNT100;
   1:  PR[GP1:91,1] = PR[GP1:90,1] + 33.318;
   1:  PR[GP1:91,2] = PR[GP1:90,2] + -5.601;
   1:L PR[91] R[100]mm/sec CNT100;
   1:  PR[GP1:91,1] = PR[GP1:90,1] + 34.056;
   1:  PR[GP1:91,2] = PR[GP1:90,2] + -0.271;
   1:L PR[91] R[100]mm/sec CNT100;
   1:  PR[GP1:91,1] = PR[GP1:90,1] + 34.040;
   1:  PR[GP1:91,2] = PR[GP1:90,2] + -0.079;
   1:L PR[91] R[100]mm/sec CNT100;
   1:  PR[GP1:91,1] = PR[GP1:90,1] + 33.310;
   1:  PR[GP1:91,2] = PR[GP1:90,2] + 5.176;
   1:L PR[91] R[100]mm/sec CNT100;
   1:  PR[GP1:91,1] = PR[GP1:90,1] + 33.282;
   1:  PR[GP1:91,2] = PR[GP1:90,2] + 5.286;
   1:L PR[91] R[100]mm/sec CNT100;
   1:  PR[GP1:91,1] = PR[GP1:90,1] + 31.027;
   1:  PR[GP1:91,2] = PR[GP1:90,2] + 10.400;
   1:L PR[91] R[100]mm/sec CNT100;
   1:  PR[GP1:91,1] = PR[GP1:90,1] + 31.005;
   1:  PR[GP1:91,2] = PR[GP1:90,2] + 10.433;
   1:L PR[91] R[100]mm/sec CNT100;
   1:  PR[GP1:91,1] = PR[GP1:90,1] + 27.406;
   1:  PR[GP1:91,2] = PR[GP1:90,2] + 14.902;
   1:L PR[91] R[100]mm/sec CNT100;
   1:  PR[GP1:91,1] = PR[GP1:90,1] + 25.636;
   1:  PR[GP1:91,2] = PR[GP1:90,2] + 16.190;
   1:L PR[91] R[100]mm/sec CNT100;
   1:  PR[GP1:91,1] = PR[GP1:90,1] + 22.698;
   1:  PR[GP1:91,2] = PR[GP1:90,2] + 18.374;
   1:L PR[91] R[100]mm/sec CNT100;
   1:  PR[GP1:91,1] = PR[GP1:90,1] + 17.199;
   1:  PR[GP1:91,2] = PR[GP1:90,2] + 20.605;
   1:L PR[91] R[100]mm/sec CNT100;
   1:  PR[GP1:91,1] = PR[GP1:90,1] + 16.735;
   1:  PR[GP1:91,2] = PR[GP1:90,2] + 20.679;
   1:L PR[91] R[100]mm/sec CNT100;
   1:  PR[GP1:91,1] = PR[GP1:90,1] + 11.294;
   1:  PR[GP1:91,2] = PR[GP1:90,2] + 21.394;
   1:L PR[91] R[100]mm/sec CNT100;
   1:  PR[GP1:91,1] = PR[GP1:90,1] + 10.386;
   1:  PR[GP1:91,2] = PR[GP1:90,2] + 21.306;
   1:L PR[91] R[100]mm/sec CNT100;
   1:  PR[GP1:91,1] = PR[GP1:90,1] + 5.339;
   1:  PR[GP1:91,2] = PR[GP1:90,2] + 20.670;
   1:L PR[91] R[100]mm/sec CNT100;
   1:  PR[GP1:91,1] = PR[GP1:90,1] + 5.047;
   1:  PR[GP1:91,2] = PR[GP1:90,2] + 20.575;
   1:L PR[91] R[100]mm/sec CNT100;
   1:  PR[GP1:91,1] = PR[GP1:90,1] + 3.442;
   1:  PR[GP1:91,2] = PR[GP1:90,2] + 19.986;
   1:L PR[91] R[100]mm/sec CNT100;
   1:  PR[GP1:91,1] = PR[GP1:90,1] + 1.226;
   1:  PR[GP1:91,2] = PR[GP1:90,2] + 19.101;
   1:L PR[91] R[100]mm/sec CNT100;
   1:  PR[GP1:91,1] = PR[GP1:90,1] + 0.926;
   1:  PR[GP1:91,2] = PR[GP1:90,2] + 19.024;
   1:L PR[91] R[100]mm/sec CNT100;
   1:  PR[GP1:91,1] = PR[GP1:90,1] + 0.534;
   1:  PR[GP1:91,2] = PR[GP1:90,2] + 18.843;
   1:L PR[91] R[100]mm/sec CNT100;
   1:  PR[91] = PR[90];
   1:  PR[GP1:91,1] = PR[GP1:90,1] + -0.986;
   1:  PR[GP1:91,2] = PR[GP1:90,2] + 19.274;
   1:  PR[GP1:91,3] = PR[GP1:90,3] + 45.445;
   1:L PR[91] R[100]mm/sec CNT100;
   1:  PR[GP1:91,1] = PR[GP1:90,1] + -2.711;
   1:  PR[GP1:91,2] = PR[GP1:90,2] + 19.963;
   1:L PR[91] R[100]mm/sec CNT100;
   1:  PR[GP1:91,1] = PR[GP1:90,1] + -4.778;
   1:  PR[GP1:91,2] = PR[GP1:90,2] + 20.717;
   1:L PR[91] R[100]mm/sec CNT100;
   1:  PR[GP1:91,1] = PR[GP1:90,1] + -4.964;
   1:  PR[GP1:91,2] = PR[GP1:90,2] + 20.776;
   1:L PR[91] R[100]mm/sec CNT100;
   1:  PR[GP1:91,1] = PR[GP1:90,1] + -9.769;
   1:  PR[GP1:91,2] = PR[GP1:90,2] + 21.380;
   1:L PR[91] R[100]mm/sec CNT100;
   1:  PR[GP1:91,1] = PR[GP1:90,1] + -10.941;
   1:  PR[GP1:91,2] = PR[GP1:90,2] + 21.493;
   1:L PR[91] R[100]mm/sec CNT100;
   1:  PR[GP1:91,1] = PR[GP1:90,1] + -16.132;
   1:  PR[GP1:91,2] = PR[GP1:90,2] + 20.811;
   1:L PR[91] R[100]mm/sec CNT100;
   1:  PR[GP1:91,1] = PR[GP1:90,1] + -16.861;
   1:  PR[GP1:91,2] = PR[GP1:90,2] + 20.695;
   1:L PR[91] R[100]mm/sec CNT100;
   1:  PR[GP1:91,1] = PR[GP1:90,1] + -22.059;
   1:  PR[GP1:91,2] = PR[GP1:90,2] + 18.590;
   1:L PR[91] R[100]mm/sec CNT100;
   1:  PR[GP1:91,1] = PR[GP1:90,1] + -22.355;
   1:  PR[GP1:91,2] = PR[GP1:90,2] + 18.460;
   1:L PR[91] R[100]mm/sec CNT100;
   1:  PR[GP1:91,1] = PR[GP1:90,1] + -27.062;
   1:  PR[GP1:91,2] = PR[GP1:90,2] + 14.958;
   1:L PR[91] R[100]mm/sec CNT100;
   1:  PR[GP1:91,1] = PR[GP1:90,1] + -28.678;
   1:  PR[GP1:91,2] = PR[GP1:90,2] + 12.917;
   1:L PR[91] R[100]mm/sec CNT100;
   1:  PR[GP1:91,1] = PR[GP1:90,1] + -30.671;
   1:  PR[GP1:91,2] = PR[GP1:90,2] + 10.441;
   1:L PR[91] R[100]mm/sec CNT100;
   1:  PR[GP1:91,1] = PR[GP1:90,1] + -32.946;
   1:  PR[GP1:91,2] = PR[GP1:90,2] + 5.252;
   1:L PR[91] R[100]mm/sec CNT100;
   1:  PR[GP1:91,1] = PR[GP1:90,1] + -33.713;
   1:  PR[GP1:91,2] = PR[GP1:90,2] + -0.353;
   1:L PR[91] R[100]mm/sec CNT100;
   1:  PR[GP1:91,1] = PR[GP1:90,1] + -33.710;
   1:  PR[GP1:91,2] = PR[GP1:90,2] + -0.395;
   1:L PR[91] R[100]mm/sec CNT100;
   1:  PR[GP1:91,1] = PR[GP1:90,1] + -32.945;
   1:  PR[GP1:91,2] = PR[GP1:90,2] + -5.878;
   1:L PR[91] R[100]mm/sec CNT100;
   1:  PR[GP1:91,1] = PR[GP1:90,1] + -32.925;
   1:  PR[GP1:91,2] = PR[GP1:90,2] + -5.924;
   1:L PR[91] R[100]mm/sec CNT100;
   1:  PR[GP1:91,1] = PR[GP1:90,1] + -30.675;
   1:  PR[GP1:91,2] = PR[GP1:90,2] + -11.053;
   1:L PR[91] R[100]mm/sec CNT100;
   1:  PR[GP1:91,1] = PR[GP1:90,1] + -27.048;
   1:  PR[GP1:91,2] = PR[GP1:90,2] + -15.596;
   1:L PR[91] R[100]mm/sec CNT100;
   1:  PR[GP1:91,1] = PR[GP1:90,1] + -22.330;
   1:  PR[GP1:91,2] = PR[GP1:90,2] + -19.099;
   1:L PR[91] R[100]mm/sec CNT100;
   1:  PR[GP1:91,1] = PR[GP1:90,1] + -22.031;
   1:  PR[GP1:91,2] = PR[GP1:90,2] + -19.229;
   1:L PR[91] R[100]mm/sec CNT100;
   1:  PR[GP1:91,1] = PR[GP1:90,1] + -16.825;
   1:  PR[GP1:91,2] = PR[GP1:90,2] + -21.328;
   1:L PR[91] R[100]mm/sec CNT100;
   1:  PR[GP1:91,1] = PR[GP1:90,1] + -16.093;
   1:  PR[GP1:91,2] = PR[GP1:90,2] + -21.444;
   1:L PR[91] R[100]mm/sec CNT100;
   1:  PR[GP1:91,1] = PR[GP1:90,1] + -10.898;
   1:  PR[GP1:91,2] = PR[GP1:90,2] + -22.117;
   1:L PR[91] R[100]mm/sec CNT100;
   1:  PR[GP1:91,1] = PR[GP1:90,1] + -9.710;
   1:  PR[GP1:91,2] = PR[GP1:90,2] + -22.000;
   1:L PR[91] R[100]mm/sec CNT100;
   1:  PR[GP1:91,1] = PR[GP1:90,1] + -4.932;
   1:  PR[GP1:91,2] = PR[GP1:90,2] + -21.389;
   1:L PR[91] R[100]mm/sec CNT100;
   1:  PR[GP1:91,1] = PR[GP1:90,1] + -3.604;
   1:  PR[GP1:91,2] = PR[GP1:90,2] + -20.926;
   1:L PR[91] R[100]mm/sec CNT100;
   1:  PR[GP1:91,1] = PR[GP1:90,1] + -0.982;
   1:  PR[GP1:91,2] = PR[GP1:90,2] + -19.898;
   1:L PR[91] R[100]mm/sec CNT100;
   1:  PR[GP1:91,1] = PR[GP1:90,1] + 0.597;
   1:  PR[GP1:91,2] = PR[GP1:90,2] + -19.657;
   1:L PR[91] R[100]mm/sec CNT100;
   1:  PR[GP1:91,1] = PR[GP1:90,1] + 0.970;
   1:  PR[GP1:91,2] = PR[GP1:90,2] + -19.857;
   1:L PR[91] R[100]mm/sec CNT100;
   1:  PR[GP1:91,1] = PR[GP1:90,1] + 1.231;
   1:  PR[GP1:91,2] = PR[GP1:90,2] + -19.935;
   1:L PR[91] R[100]mm/sec CNT100;
   1:  PR[GP1:91,1] = PR[GP1:90,1] + 3.761;
   1:  PR[GP1:91,2] = PR[GP1:90,2] + -20.926;
   1:L PR[91] R[100]mm/sec CNT100;
   1:  PR[GP1:91,1] = PR[GP1:90,1] + 4.933;
   1:  PR[GP1:91,2] = PR[GP1:90,2] + -21.338;
   1:L PR[91] R[100]mm/sec CNT100;
   1:  PR[GP1:91,1] = PR[GP1:90,1] + 9.660;
   1:  PR[GP1:91,2] = PR[GP1:90,2] + -21.950;
   1:L PR[91] R[100]mm/sec CNT100;
   1:  PR[GP1:91,1] = PR[GP1:90,1] + 9.924;
   1:  PR[GP1:91,2] = PR[GP1:90,2] + -22.006;
   1:L PR[91] R[100]mm/sec CNT100;
   1:  PR[GP1:91,1] = PR[GP1:90,1] + 11.053;
   1:  PR[GP1:91,2] = PR[GP1:90,2] + -22.117;
   1:L PR[91] R[100]mm/sec CNT100;
   1:  PR[GP1:91,1] = PR[GP1:90,1] + 16.248;
   1:  PR[GP1:91,2] = PR[GP1:90,2] + -21.444;
   1:L PR[91] R[100]mm/sec CNT100;
   1:  PR[GP1:91,1] = PR[GP1:90,1] + 16.980;
   1:  PR[GP1:91,2] = PR[GP1:90,2] + -21.328;
   1:L PR[91] R[100]mm/sec CNT100;
   1:  PR[GP1:91,1] = PR[GP1:90,1] + 22.187;
   1:  PR[GP1:91,2] = PR[GP1:90,2] + -19.230;
   1:L PR[91] R[100]mm/sec CNT100;
   1:  PR[GP1:91,1] = PR[GP1:90,1] + 22.485;
   1:  PR[GP1:91,2] = PR[GP1:90,2] + -19.101;
   1:L PR[91] R[100]mm/sec CNT100;
   1:  PR[GP1:91,1] = PR[GP1:90,1] + 27.203;
   1:  PR[GP1:91,2] = PR[GP1:90,2] + -15.598;
   1:L PR[91] R[100]mm/sec CNT100;
   1:  PR[GP1:91,1] = PR[GP1:90,1] + 30.831;
   1:  PR[GP1:91,2] = PR[GP1:90,2] + -11.046;
   1:L PR[91] R[100]mm/sec CNT100;
   1:  PR[GP1:91,1] = PR[GP1:90,1] + 33.101;
   1:  PR[GP1:91,2] = PR[GP1:90,2] + -5.900;
   1:L PR[91] R[100]mm/sec CNT100;
   1:  PR[GP1:91,1] = PR[GP1:90,1] + 33.870;
   1:  PR[GP1:91,2] = PR[GP1:90,2] + -0.273;
   1:L PR[91] R[100]mm/sec CNT100;
   1:  PR[GP1:91,1] = PR[GP1:90,1] + 33.866;
   1:  PR[GP1:91,2] = PR[GP1:90,2] + -0.223;
   1:L PR[91] R[100]mm/sec CNT100;
   1:  PR[GP1:91,1] = PR[GP1:90,1] + 33.103;
   1:  PR[GP1:91,2] = PR[GP1:90,2] + 5.269;
   1:L PR[91] R[100]mm/sec CNT100;
   1:  PR[GP1:91,1] = PR[GP1:90,1] + 30.838;
   1:  PR[GP1:91,2] = PR[GP1:90,2] + 10.410;
   1:L PR[91] R[100]mm/sec CNT100;
   1:  PR[GP1:91,1] = PR[GP1:90,1] + 27.219;
   1:  PR[GP1:91,2] = PR[GP1:90,2] + 14.959;
   1:L PR[91] R[100]mm/sec CNT100;
   1:  PR[GP1:91,1] = PR[GP1:90,1] + 22.510;
   1:  PR[GP1:91,2] = PR[GP1:90,2] + 18.463;
   1:L PR[91] R[100]mm/sec CNT100;
   1:  PR[GP1:91,1] = PR[GP1:90,1] + 22.214;
   1:  PR[GP1:91,2] = PR[GP1:90,2] + 18.592;
   1:L PR[91] R[100]mm/sec CNT100;
   1:  PR[GP1:91,1] = PR[GP1:90,1] + 17.015;
   1:  PR[GP1:91,2] = PR[GP1:90,2] + 20.694;
   1:L PR[91] R[100]mm/sec CNT100;
   1:  PR[GP1:91,1] = PR[GP1:90,1] + 16.286;
   1:  PR[GP1:91,2] = PR[GP1:90,2] + 20.811;
   1:L PR[91] R[100]mm/sec CNT100;
   1:  PR[GP1:91,1] = PR[GP1:90,1] + 11.095;
   1:  PR[GP1:91,2] = PR[GP1:90,2] + 21.493;
   1:L PR[91] R[100]mm/sec CNT100;
   1:  PR[GP1:91,1] = PR[GP1:90,1] + 9.923;
   1:  PR[GP1:91,2] = PR[GP1:90,2] + 21.380;
   1:L PR[91] R[100]mm/sec CNT100;
   1:  PR[GP1:91,1] = PR[GP1:90,1] + 5.122;
   1:  PR[GP1:91,2] = PR[GP1:90,2] + 20.775;
   1:L PR[91] R[100]mm/sec CNT100;
   1:  PR[GP1:91,1] = PR[GP1:90,1] + 4.754;
   1:  PR[GP1:91,2] = PR[GP1:90,2] + 20.655;
   1:L PR[91] R[100]mm/sec CNT100;
   1:  PR[GP1:91,1] = PR[GP1:90,1] + 2.867;
   1:  PR[GP1:91,2] = PR[GP1:90,2] + 19.962;
   1:L PR[91] R[100]mm/sec CNT100;
   1:  PR[GP1:91,1] = PR[GP1:90,1] + 1.209;
   1:  PR[GP1:91,2] = PR[GP1:90,2] + 19.301;
   1:L PR[91] R[100]mm/sec CNT100;
   1:  PR[GP1:91,1] = PR[GP1:90,1] + 0.997;
   1:  PR[GP1:91,2] = PR[GP1:90,2] + 19.246;
   1:L PR[91] R[100]mm/sec CNT100;
   1:  PR[GP1:91,1] = PR[GP1:90,1] + 0.550;
   1:  PR[GP1:91,2] = PR[GP1:90,2] + 19.040;
   1:L PR[91] R[100]mm/sec CNT100;
   1:  PR[91] = PR[90];
   1:  PR[GP1:91,1] = PR[GP1:90,1] + -0.971;
   1:  PR[GP1:91,2] = PR[GP1:90,2] + 19.474;
   1:  PR[GP1:91,3] = PR[GP1:90,3] + 46.055;
   1:L PR[91] R[100]mm/sec CNT100;
   1:  PR[GP1:91,1] = PR[GP1:90,1] + -2.135;
   1:  PR[GP1:91,2] = PR[GP1:90,2] + 19.940;
   1:L PR[91] R[100]mm/sec CNT100;
   1:  PR[GP1:91,1] = PR[GP1:90,1] + -4.511;
   1:  PR[GP1:91,2] = PR[GP1:90,2] + 20.806;
   1:L PR[91] R[100]mm/sec CNT100;
   1:  PR[GP1:91,1] = PR[GP1:90,1] + -4.747;
   1:  PR[GP1:91,2] = PR[GP1:90,2] + 20.881;
   1:L PR[91] R[100]mm/sec CNT100;
   1:  PR[GP1:91,1] = PR[GP1:90,1] + -9.306;
   1:  PR[GP1:91,2] = PR[GP1:90,2] + 21.454;
   1:L PR[91] R[100]mm/sec CNT100;
   1:  PR[GP1:91,1] = PR[GP1:90,1] + -10.742;
   1:  PR[GP1:91,2] = PR[GP1:90,2] + 21.593;
   1:L PR[91] R[100]mm/sec CNT100;
   1:  PR[GP1:91,1] = PR[GP1:90,1] + -15.682;
   1:  PR[GP1:91,2] = PR[GP1:90,2] + 20.944;
   1:L PR[91] R[100]mm/sec CNT100;
   1:  PR[GP1:91,1] = PR[GP1:90,1] + -16.676;
   1:  PR[GP1:91,2] = PR[GP1:90,2] + 20.784;
   1:L PR[91] R[100]mm/sec CNT100;
   1:  PR[GP1:91,1] = PR[GP1:90,1] + -21.635;
   1:  PR[GP1:91,2] = PR[GP1:90,2] + 18.777;
   1:L PR[91] R[100]mm/sec CNT100;
   1:  PR[GP1:91,1] = PR[GP1:90,1] + -22.182;
   1:  PR[GP1:91,2] = PR[GP1:90,2] + 18.538;
   1:L PR[91] R[100]mm/sec CNT100;
   1:  PR[GP1:91,1] = PR[GP1:90,1] + -26.899;
   1:  PR[GP1:91,2] = PR[GP1:90,2] + 15.020;
   1:L PR[91] R[100]mm/sec CNT100;
   1:  PR[GP1:91,1] = PR[GP1:90,1] + -30.490;
   1:  PR[GP1:91,2] = PR[GP1:90,2] + 10.479;
   1:L PR[91] R[100]mm/sec CNT100;
   1:  PR[GP1:91,1] = PR[GP1:90,1] + -32.742;
   1:  PR[GP1:91,2] = PR[GP1:90,2] + 5.296;
   1:L PR[91] R[100]mm/sec CNT100;
   1:  PR[GP1:91,1] = PR[GP1:90,1] + -33.521;
   1:  PR[GP1:91,2] = PR[GP1:90,2] + -0.312;
   1:L PR[91] R[100]mm/sec CNT100;
   1:  PR[GP1:91,1] = PR[GP1:90,1] + -32.746;
   1:  PR[GP1:91,2] = PR[GP1:90,2] + -5.914;
   1:L PR[91] R[100]mm/sec CNT100;
   1:  PR[GP1:91,1] = PR[GP1:90,1] + -30.483;
   1:  PR[GP1:91,2] = PR[GP1:90,2] + -11.116;
   1:L PR[91] R[100]mm/sec CNT100;
   1:  PR[GP1:91,1] = PR[GP1:90,1] + -26.883;
   1:  PR[GP1:91,2] = PR[GP1:90,2] + -15.659;
   1:L PR[91] R[100]mm/sec CNT100;
   1:  PR[GP1:91,1] = PR[GP1:90,1] + -22.157;
   1:  PR[GP1:91,2] = PR[GP1:90,2] + -19.176;
   1:L PR[91] R[100]mm/sec CNT100;
   1:  PR[GP1:91,1] = PR[GP1:90,1] + -21.607;
   1:  PR[GP1:91,2] = PR[GP1:90,2] + -19.415;
   1:L PR[91] R[100]mm/sec CNT100;
   1:  PR[GP1:91,1] = PR[GP1:90,1] + -16.641;
   1:  PR[GP1:91,2] = PR[GP1:90,2] + -21.418;
   1:L PR[91] R[100]mm/sec CNT100;
   1:  PR[GP1:91,1] = PR[GP1:90,1] + -15.644;
   1:  PR[GP1:91,2] = PR[GP1:90,2] + -21.576;
   1:L PR[91] R[100]mm/sec CNT100;
   1:  PR[GP1:91,1] = PR[GP1:90,1] + -10.699;
   1:  PR[GP1:91,2] = PR[GP1:90,2] + -22.217;
   1:L PR[91] R[100]mm/sec CNT100;
   1:  PR[GP1:91,1] = PR[GP1:90,1] + -9.246;
   1:  PR[GP1:91,2] = PR[GP1:90,2] + -22.073;
   1:L PR[91] R[100]mm/sec CNT100;
   1:  PR[GP1:91,1] = PR[GP1:90,1] + -4.716;
   1:  PR[GP1:91,2] = PR[GP1:90,2] + -21.494;
   1:L PR[91] R[100]mm/sec CNT100;
   1:  PR[GP1:91,1] = PR[GP1:90,1] + -3.169;
   1:  PR[GP1:91,2] = PR[GP1:90,2] + -20.955;
   1:L PR[91] R[100]mm/sec CNT100;
   1:  PR[GP1:91,1] = PR[GP1:90,1] + -0.976;
   1:  PR[GP1:91,2] = PR[GP1:90,2] + -20.095;
   1:L PR[91] R[100]mm/sec CNT100;
   1:  PR[GP1:91,1] = PR[GP1:90,1] + -0.287;
   1:  PR[GP1:91,2] = PR[GP1:90,2] + -19.979;
   1:L PR[91] R[100]mm/sec CNT100;
   1:  PR[GP1:91,1] = PR[GP1:90,1] + 0.634;
   1:  PR[GP1:91,2] = PR[GP1:90,2] + -19.864;
   1:L PR[91] R[100]mm/sec CNT100;
   1:  PR[GP1:91,1] = PR[GP1:90,1] + 1.011;
   1:  PR[GP1:91,2] = PR[GP1:90,2] + -20.067;
   1:L PR[91] R[100]mm/sec CNT100;
   1:  PR[GP1:91,1] = PR[GP1:90,1] + 1.215;
   1:  PR[GP1:91,2] = PR[GP1:90,2] + -20.128;
   1:L PR[91] R[100]mm/sec CNT100;
   1:  PR[GP1:91,1] = PR[GP1:90,1] + 3.327;
   1:  PR[GP1:91,2] = PR[GP1:90,2] + -20.955;
   1:L PR[91] R[100]mm/sec CNT100;
   1:  PR[GP1:91,1] = PR[GP1:90,1] + 4.694;
   1:  PR[GP1:91,2] = PR[GP1:90,2] + -21.436;
   1:L PR[91] R[100]mm/sec CNT100;
   1:  PR[GP1:91,1] = PR[GP1:90,1] + 9.140;
   1:  PR[GP1:91,2] = PR[GP1:90,2] + -22.011;
   1:L PR[91] R[100]mm/sec CNT100;
   1:  PR[GP1:91,1] = PR[GP1:90,1] + 9.459;
   1:  PR[GP1:91,2] = PR[GP1:90,2] + -22.079;
   1:L PR[91] R[100]mm/sec CNT100;
   1:  PR[GP1:91,1] = PR[GP1:90,1] + 10.854;
   1:  PR[GP1:91,2] = PR[GP1:90,2] + -22.217;
   1:L PR[91] R[100]mm/sec CNT100;
   1:  PR[GP1:91,1] = PR[GP1:90,1] + 15.799;
   1:  PR[GP1:91,2] = PR[GP1:90,2] + -21.576;
   1:L PR[91] R[100]mm/sec CNT100;
   1:  PR[GP1:91,1] = PR[GP1:90,1] + 16.796;
   1:  PR[GP1:91,2] = PR[GP1:90,2] + -21.417;
   1:L PR[91] R[100]mm/sec CNT100;
   1:  PR[GP1:91,1] = PR[GP1:90,1] + 21.763;
   1:  PR[GP1:91,2] = PR[GP1:90,2] + -19.417;
   1:L PR[91] R[100]mm/sec CNT100;
   1:  PR[GP1:91,1] = PR[GP1:90,1] + 22.312;
   1:  PR[GP1:91,2] = PR[GP1:90,2] + -19.178;
   1:L PR[91] R[100]mm/sec CNT100;
   1:  PR[GP1:91,1] = PR[GP1:90,1] + 27.038;
   1:  PR[GP1:91,2] = PR[GP1:90,2] + -15.661;
   1:L PR[91] R[100]mm/sec CNT100;
   1:  PR[GP1:91,1] = PR[GP1:90,1] + 30.639;
   1:  PR[GP1:91,2] = PR[GP1:90,2] + -11.108;
   1:L PR[91] R[100]mm/sec CNT100;
   1:  PR[GP1:91,1] = PR[GP1:90,1] + 32.896;
   1:  PR[GP1:91,2] = PR[GP1:90,2] + -5.943;
   1:L PR[91] R[100]mm/sec CNT100;
   1:  PR[GP1:91,1] = PR[GP1:90,1] + 33.681;
   1:  PR[GP1:91,2] = PR[GP1:90,2] + -0.291;
   1:L PR[91] R[100]mm/sec CNT100;
   1:  PR[GP1:91,1] = PR[GP1:90,1] + 32.899;
   1:  PR[GP1:91,2] = PR[GP1:90,2] + 5.312;
   1:L PR[91] R[100]mm/sec CNT100;
   1:  PR[GP1:91,1] = PR[GP1:90,1] + 30.647;
   1:  PR[GP1:91,2] = PR[GP1:90,2] + 10.472;
   1:L PR[91] R[100]mm/sec CNT100;
   1:  PR[GP1:91,1] = PR[GP1:90,1] + 27.054;
   1:  PR[GP1:91,2] = PR[GP1:90,2] + 15.022;
   1:L PR[91] R[100]mm/sec CNT100;
   1:  PR[GP1:91,1] = PR[GP1:90,1] + 22.338;
   1:  PR[GP1:91,2] = PR[GP1:90,2] + 18.540;
   1:L PR[91] R[100]mm/sec CNT100;
   1:  PR[GP1:91,1] = PR[GP1:90,1] + 21.790;
   1:  PR[GP1:91,2] = PR[GP1:90,2] + 18.779;
   1:L PR[91] R[100]mm/sec CNT100;
   1:  PR[GP1:91,1] = PR[GP1:90,1] + 16.831;
   1:  PR[GP1:91,2] = PR[GP1:90,2] + 20.784;
   1:L PR[91] R[100]mm/sec CNT100;
   1:  PR[GP1:91,1] = PR[GP1:90,1] + 15.836;
   1:  PR[GP1:91,2] = PR[GP1:90,2] + 20.944;
   1:L PR[91] R[100]mm/sec CNT100;
   1:  PR[GP1:91,1] = PR[GP1:90,1] + 10.896;
   1:  PR[GP1:91,2] = PR[GP1:90,2] + 21.593;
   1:L PR[91] R[100]mm/sec CNT100;
   1:  PR[GP1:91,1] = PR[GP1:90,1] + 9.460;
   1:  PR[GP1:91,2] = PR[GP1:90,2] + 21.454;
   1:L PR[91] R[100]mm/sec CNT100;
   1:  PR[GP1:91,1] = PR[GP1:90,1] + 4.906;
   1:  PR[GP1:91,2] = PR[GP1:90,2] + 20.880;
   1:L PR[91] R[100]mm/sec CNT100;
   1:  PR[GP1:91,1] = PR[GP1:90,1] + 4.461;
   1:  PR[GP1:91,2] = PR[GP1:90,2] + 20.735;
   1:L PR[91] R[100]mm/sec CNT100;
   1:  PR[GP1:91,1] = PR[GP1:90,1] + 2.292;
   1:  PR[GP1:91,2] = PR[GP1:90,2] + 19.939;
   1:L PR[91] R[100]mm/sec CNT100;
